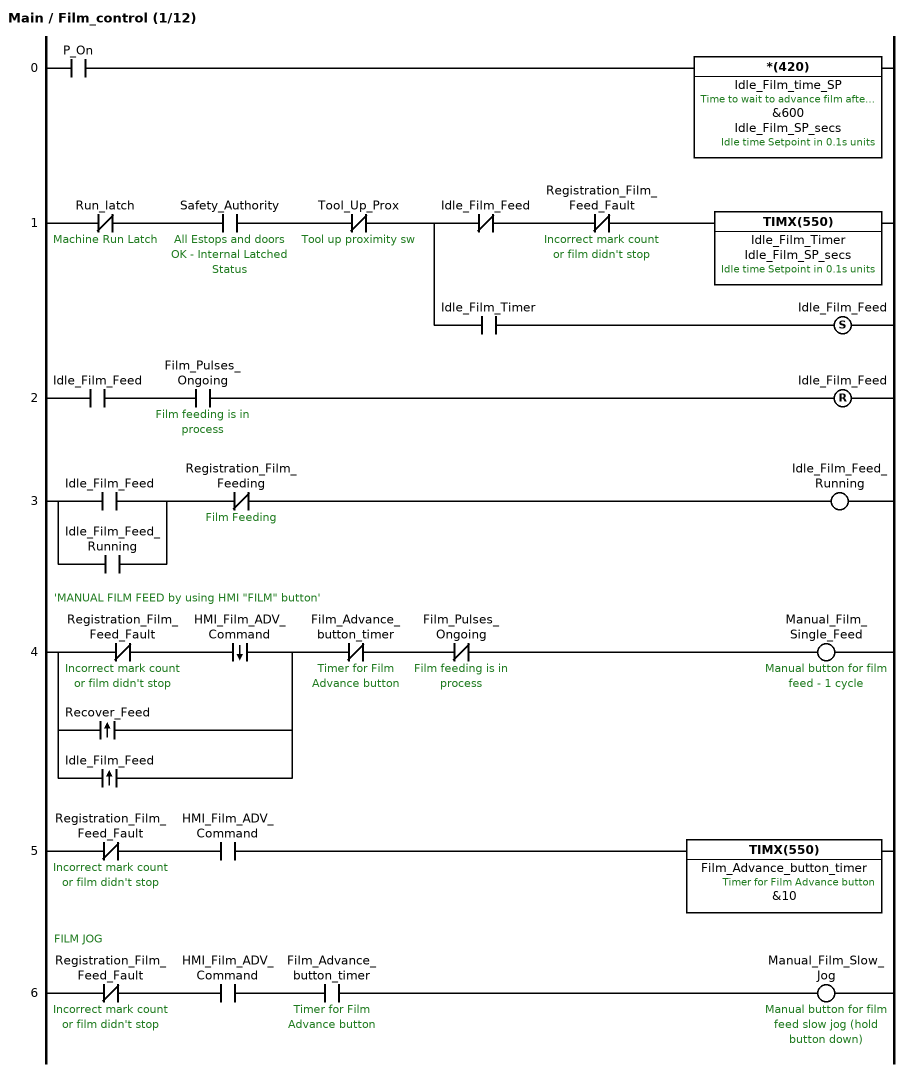
; [picture p72: Main / Film_control, rungs 0-6]
; rung 0
LD P_On
*(420) Idle_Film_time_SP &600 Idle_Film_SP_secs  ; Time to wait to advance film after sitting idle in minutes, Idle time Setpoint in 0.1s units
; rung 1
LDNOT Run_latch  ; Machine Run Latch
AND Safety_Authority  ; All Estops and doors OK - Internal Latched Status
ANDNOT Tool_Up_Prox  ; Tool up proximity sw
OUT TR0
ANDNOT Idle_Film_Feed
ANDNOT Registration_Film_Feed_Fault  ; Incorrect mark count or film didn't stop
TIMX(550) Idle_Film_Timer Idle_Film_SP_secs  ; Idle time Setpoint in 0.1s units
LD TR0
AND Idle_Film_Timer
SET Idle_Film_Feed
; rung 2
LD Idle_Film_Feed
AND Film_Pulses_Ongoing  ; Film feeding is in process
RSET Idle_Film_Feed
; rung 3
LD Idle_Film_Feed
OR Idle_Film_Feed_Running
ANDNOT Registration_Film_Feeding  ; Film Feeding
OUT Idle_Film_Feed_Running
; rung 4: 'MANUAL FILM FEED by using HMI "FILM" button'
LDNOT Registration_Film_Feed_Fault  ; Incorrect mark count or film didn't stop
%AND HMI_Film_ADV_Command
@OR Recover_Feed
@OR Idle_Film_Feed
ANDNOT Film_Advance_button_timer  ; Timer for Film Advance button
ANDNOT Film_Pulses_Ongoing  ; Film feeding is in process
OUT Manual_Film_Single_Feed  ; Manual button for film feed - 1 cycle
; rung 5
LDNOT Registration_Film_Feed_Fault  ; Incorrect mark count or film didn't stop
AND HMI_Film_ADV_Command
TIMX(550) Film_Advance_button_timer &10  ; Timer for Film Advance button
; rung 6: FILM JOG
LDNOT Registration_Film_Feed_Fault  ; Incorrect mark count or film didn't stop
AND HMI_Film_ADV_Command
AND Film_Advance_button_timer  ; Timer for Film Advance button
OUT Manual_Film_Slow_Jog  ; Manual button for film feed slow jog (hold button down)

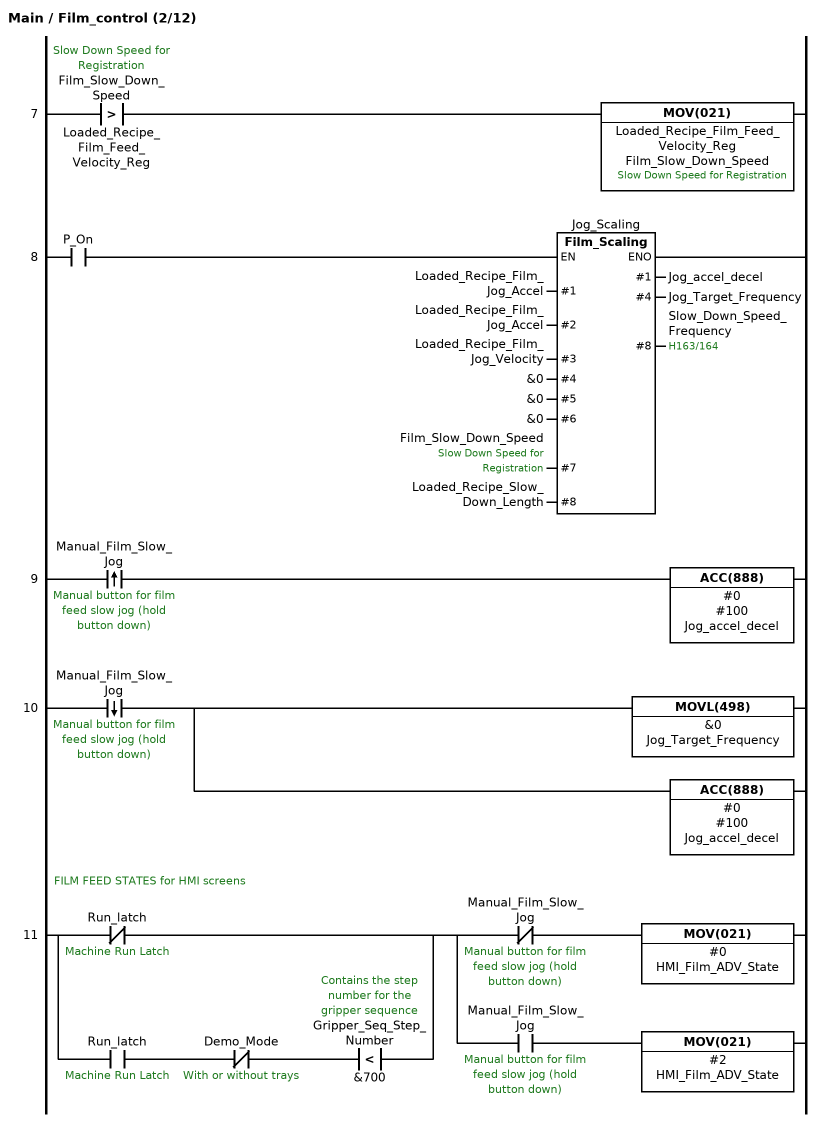
; rung 7
LD>(320) Film_Slow_Down_Speed Loaded_Recipe_Film_Feed_Velocity_Reg  ; Slow Down Speed for Registration
MOV(021) Loaded_Recipe_Film_Feed_Velocity_Reg Film_Slow_Down_Speed  ; Slow Down Speed for Registration
; rung 8
LD P_On
CALL Jog_Scaling : Film_Scaling (#1 := Loaded_Recipe_Film_Jog_Accel, #2 := Loaded_Recipe_Film_Jog_Accel, #3 := Loaded_Recipe_Film_Jog_Velocity, #4 := &0, #5 := &0, #6 := &0, #7 := Film_Slow_Down_Speed, #8 := Loaded_Recipe_Slow_Down_Length)  ; Slow Down Speed for Registration, H163/164
; rung 9
@LD Manual_Film_Slow_Jog  ; Manual button for film feed slow jog (hold button down)
ACC(888) #0 #100 Jog_accel_decel
; rung 10
%LD Manual_Film_Slow_Jog  ; Manual button for film feed slow jog (hold button down)
MOVL(498) &0 Jog_Target_Frequency
ACC(888) #0 #100 Jog_accel_decel
; rung 11: FILM FEED STATES for HMI screens
LDNOT Run_latch  ; Machine Run Latch
LD Run_latch  ; Machine Run Latch
ANDNOT Demo_Mode  ; With or without trays
AND<(310) Gripper_Seq_Step_Number &700  ; Contains the step number for the gripper sequence
ORLD
OUT TR0
ANDNOT Manual_Film_Slow_Jog  ; Manual button for film feed slow jog (hold button down)
MOV(021) #0 HMI_Film_ADV_State
LD TR0
AND Manual_Film_Slow_Jog  ; Manual button for film feed slow jog (hold button down)
MOV(021) #2 HMI_Film_ADV_State

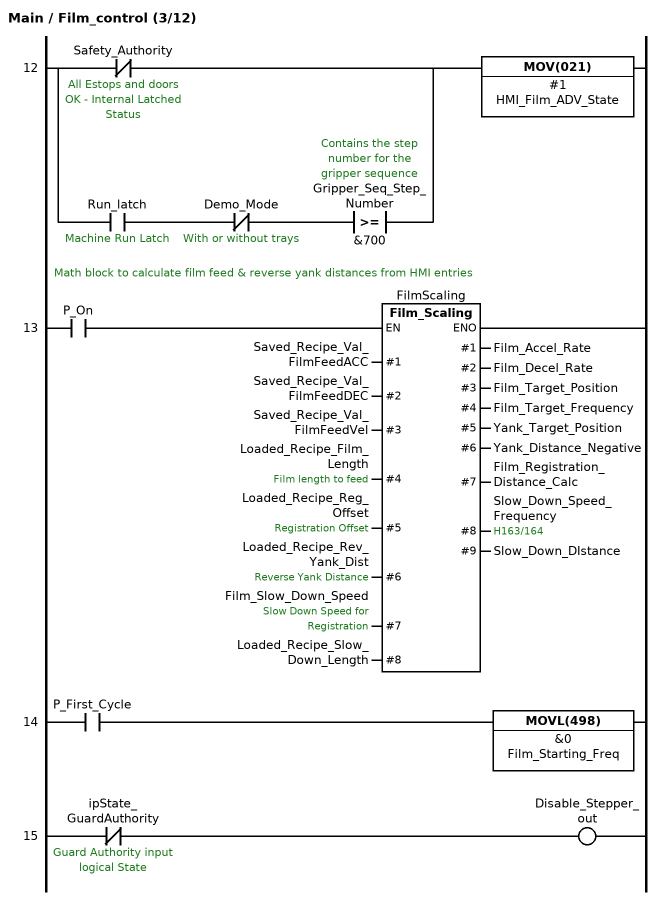
; rung 12
LDNOT Safety_Authority  ; All Estops and doors OK - Internal Latched Status
LD Run_latch  ; Machine Run Latch
ANDNOT Demo_Mode  ; With or without trays
AND>=(325) Gripper_Seq_Step_Number &700  ; Contains the step number for the gripper sequence
ORLD
MOV(021) #1 HMI_Film_ADV_State
; rung 13: Math block to calculate film feed & reverse yank distances from HMI entries
LD P_On
CALL FilmScaling : Film_Scaling (#1 := Saved_Recipe_Val_FilmFeedACC, #2 := Saved_Recipe_Val_FilmFeedDEC, #3 := Saved_Recipe_Val_FilmFeedVel, #4 := Loaded_Recipe_Film_Length, #5 := Loaded_Recipe_Reg_Offset, #6 := Loaded_Recipe_Rev_Yank_Dist, #7 := Film_Slow_Down_Speed, #8 := Loaded_Recipe_Slow_Down_Length, #9 => Slow_Down_DIstance)  ; Film length to feed, Registration Offset, Reverse Yank Distance, Slow Down Speed for Registration, H163/164
; rung 14
LD P_First_Cycle
MOVL(498) &0 Film_Starting_Freq
; rung 15
LDNOT ipState_GuardAuthority  ; Guard Authority input logical State
OUT Disable_Stepper_out

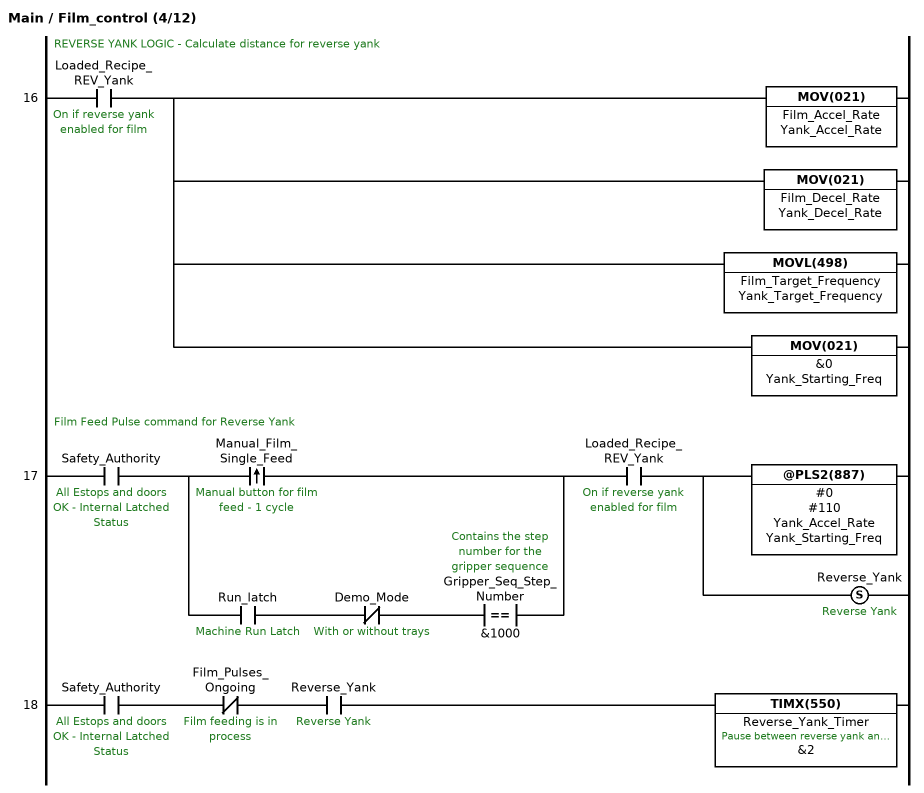
; rung 16: REVERSE YANK LOGIC - Calculate distance for reverse yank
LD Loaded_Recipe_REV_Yank  ; On if reverse yank enabled for film
MOV(021) Film_Accel_Rate Yank_Accel_Rate
MOV(021) Film_Decel_Rate Yank_Decel_Rate
MOVL(498) Film_Target_Frequency Yank_Target_Frequency
MOV(021) &0 Yank_Starting_Freq
; rung 17: Film Feed Pulse command for Reverse Yank
LD Safety_Authority  ; All Estops and doors OK - Internal Latched Status
@LD Manual_Film_Single_Feed  ; Manual button for film feed - 1 cycle
LD Run_latch  ; Machine Run Latch
ANDNOT Demo_Mode  ; With or without trays
AND=(300) Gripper_Seq_Step_Number &1000  ; Contains the step number for the gripper sequence
ORLD
ANDLD
AND Loaded_Recipe_REV_Yank  ; On if reverse yank enabled for film
@PLS2(887) #0 #110 Yank_Accel_Rate Yank_Starting_Freq
SET Reverse_Yank  ; Reverse Yank
; rung 18
LD Safety_Authority  ; All Estops and doors OK - Internal Latched Status
ANDNOT Film_Pulses_Ongoing  ; Film feeding is in process
AND Reverse_Yank  ; Reverse Yank
TIMX(550) Reverse_Yank_Timer &2  ; Pause between reverse yank and moving forward

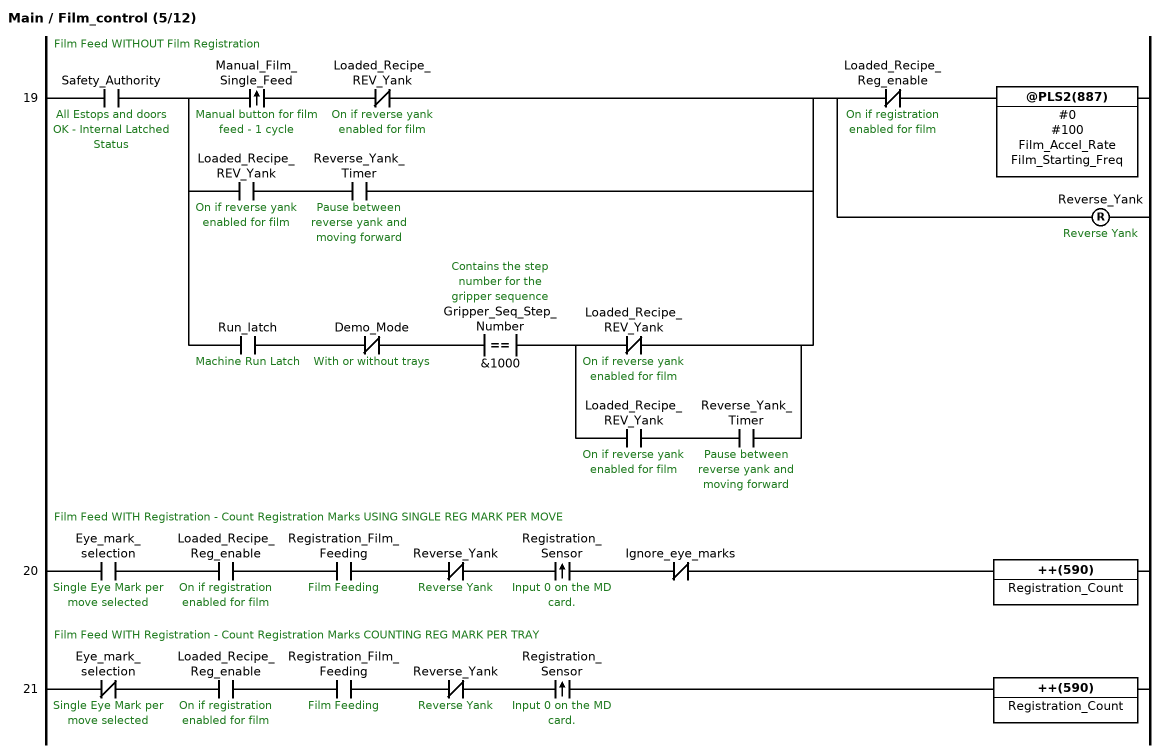
; rung 19: Film Feed WITHOUT Film Registration
LD Safety_Authority  ; All Estops and doors OK - Internal Latched Status
@LD Manual_Film_Single_Feed  ; Manual button for film feed - 1 cycle
ANDNOT Loaded_Recipe_REV_Yank  ; On if reverse yank enabled for film
LD Loaded_Recipe_REV_Yank  ; On if reverse yank enabled for film
AND Reverse_Yank_Timer  ; Pause between reverse yank and moving forward
ORLD
LD Run_latch  ; Machine Run Latch
ANDNOT Demo_Mode  ; With or without trays
AND=(300) Gripper_Seq_Step_Number &1000  ; Contains the step number for the gripper sequence
LDNOT Loaded_Recipe_REV_Yank  ; On if reverse yank enabled for film
LD Loaded_Recipe_REV_Yank  ; On if reverse yank enabled for film
AND Reverse_Yank_Timer  ; Pause between reverse yank and moving forward
ORLD
ANDLD
ORLD
ANDLD
OUT TR0
ANDNOT Loaded_Recipe_Reg_enable  ; On if registration enabled for film
@PLS2(887) #0 #100 Film_Accel_Rate Film_Starting_Freq
LD TR0
RSET Reverse_Yank  ; Reverse Yank
; rung 20: Film Feed WITH Registration - Count Registration Marks USING SINGLE REG MARK PER MOVE
LD Eye_mark_selection  ; Single Eye Mark per move selected
AND Loaded_Recipe_Reg_enable  ; On if registration enabled for film
AND Registration_Film_Feeding  ; Film Feeding
ANDNOT Reverse_Yank  ; Reverse Yank
@AND Registration_Sensor  ; Input 0 on the MD card.
ANDNOT Ignore_eye_marks
++(590) Registration_Count
; rung 21: Film Feed WITH Registration - Count Registration Marks COUNTING REG MARK PER TRAY
LDNOT Eye_mark_selection  ; Single Eye Mark per move selected
AND Loaded_Recipe_Reg_enable  ; On if registration enabled for film
AND Registration_Film_Feeding  ; Film Feeding
ANDNOT Reverse_Yank  ; Reverse Yank
@AND Registration_Sensor  ; Input 0 on the MD card.
++(590) Registration_Count

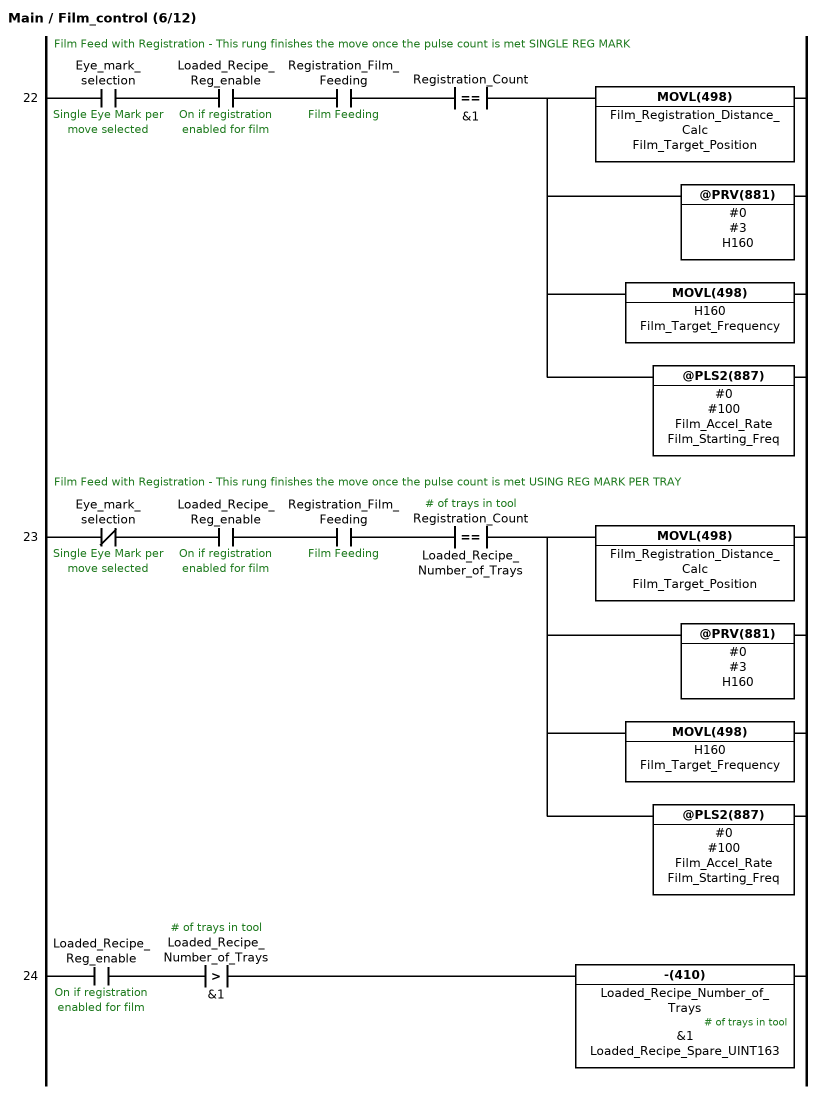
; rung 22: Film Feed with Registration - This rung finishes the move once the pulse count is met SINGLE REG MARK
LD Eye_mark_selection  ; Single Eye Mark per move selected
AND Loaded_Recipe_Reg_enable  ; On if registration enabled for film
AND Registration_Film_Feeding  ; Film Feeding
AND=(300) Registration_Count &1
MOVL(498) Film_Registration_Distance_Calc Film_Target_Position
@PRV(881) #0 #3 H160
MOVL(498) H160 Film_Target_Frequency
@PLS2(887) #0 #100 Film_Accel_Rate Film_Starting_Freq
; rung 23: Film Feed with Registration - This rung finishes the move once the pulse count is met USING REG MARK PER TRAY
LDNOT Eye_mark_selection  ; Single Eye Mark per move selected
AND Loaded_Recipe_Reg_enable  ; On if registration enabled for film
AND Registration_Film_Feeding  ; Film Feeding
AND=(300) Registration_Count Loaded_Recipe_Number_of_Trays  ; # of trays in tool
MOVL(498) Film_Registration_Distance_Calc Film_Target_Position
@PRV(881) #0 #3 H160
MOVL(498) H160 Film_Target_Frequency
@PLS2(887) #0 #100 Film_Accel_Rate Film_Starting_Freq
; rung 24
LD Loaded_Recipe_Reg_enable  ; On if registration enabled for film
AND>(320) Loaded_Recipe_Number_of_Trays &1  ; # of trays in tool
-(410) Loaded_Recipe_Number_of_Trays &1 Loaded_Recipe_Spare_UINT163  ; # of trays in tool

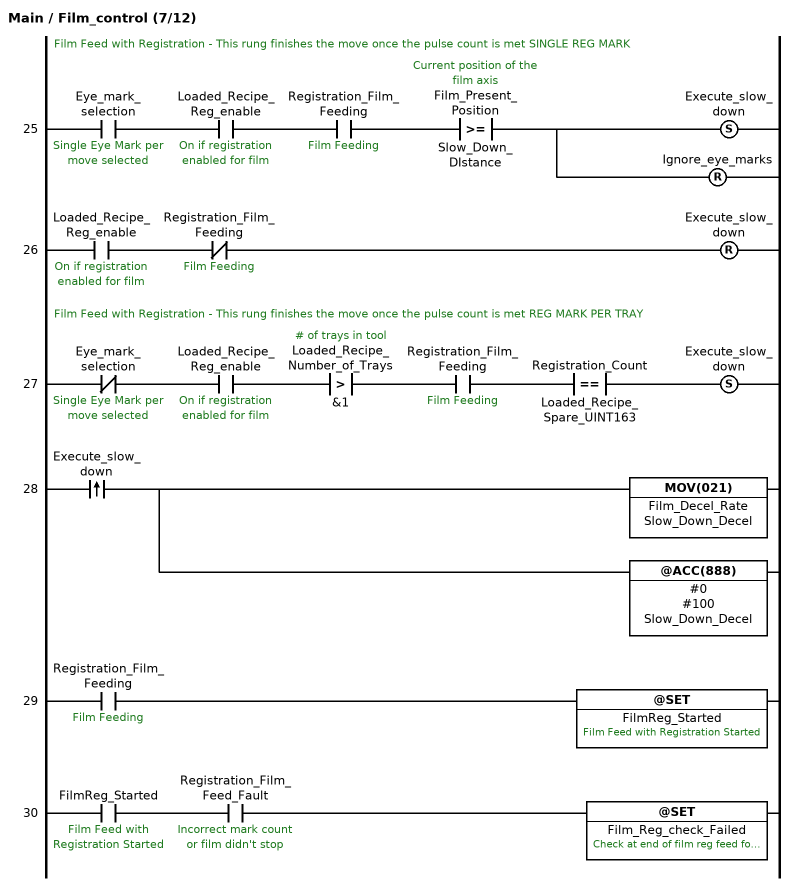
; rung 25: Film Feed with Registration - This rung finishes the move once the pulse count is met SINGLE REG MARK
LD Eye_mark_selection  ; Single Eye Mark per move selected
AND Loaded_Recipe_Reg_enable  ; On if registration enabled for film
AND Registration_Film_Feeding  ; Film Feeding
AND>=(325) Film_Present_Position Slow_Down_DIstance  ; Current position of the film axis
SET Execute_slow_down
RSET Ignore_eye_marks
; rung 26
LD Loaded_Recipe_Reg_enable  ; On if registration enabled for film
ANDNOT Registration_Film_Feeding  ; Film Feeding
RSET Execute_slow_down
; rung 27: Film Feed with Registration - This rung finishes the move once the pulse count is met REG MARK PER TRAY
LDNOT Eye_mark_selection  ; Single Eye Mark per move selected
AND Loaded_Recipe_Reg_enable  ; On if registration enabled for film
AND>(320) Loaded_Recipe_Number_of_Trays &1  ; # of trays in tool
AND Registration_Film_Feeding  ; Film Feeding
AND=(300) Registration_Count Loaded_Recipe_Spare_UINT163
SET Execute_slow_down
; rung 28
@LD Execute_slow_down
MOV(021) Film_Decel_Rate Slow_Down_Decel
@ACC(888) #0 #100 Slow_Down_Decel
; rung 29
LD Registration_Film_Feeding  ; Film Feeding
@SET FilmReg_Started  ; Film Feed with Registration Started
; rung 30
LD FilmReg_Started  ; Film Feed with Registration Started
AND Registration_Film_Feed_Fault  ; Incorrect mark count or film didn't stop
@SET Film_Reg_check_Failed  ; Check at end of film reg feed for problems

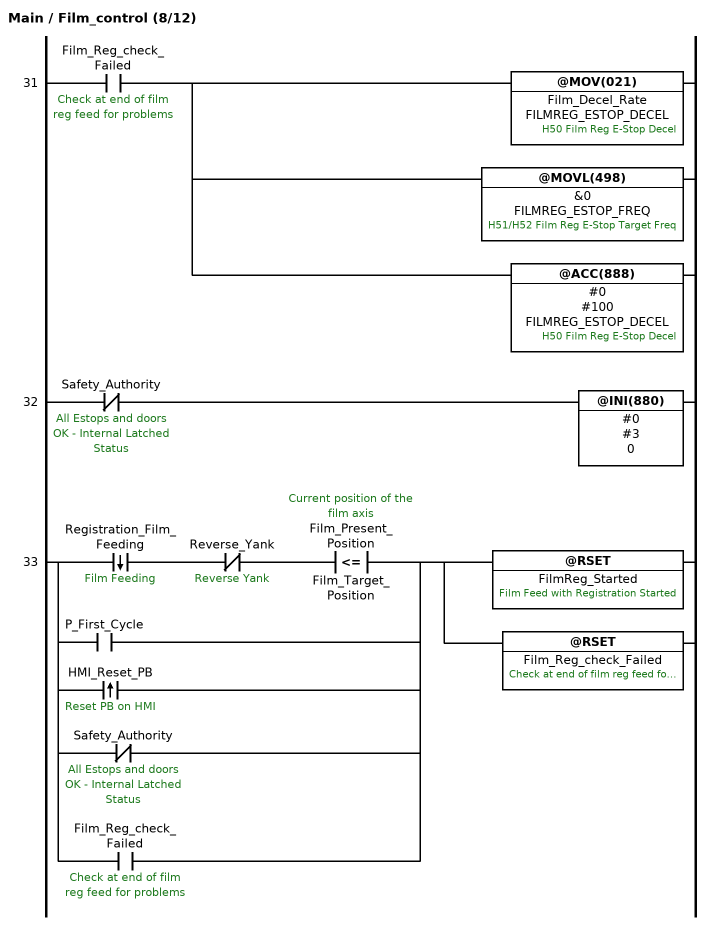
; rung 31
LD Film_Reg_check_Failed  ; Check at end of film reg feed for problems
@MOV(021) Film_Decel_Rate FILMREG_ESTOP_DECEL  ; H50 Film Reg E-Stop Decel
@MOVL(498) &0 FILMREG_ESTOP_FREQ  ; H51/H52 Film Reg E-Stop Target Freq
@ACC(888) #0 #100 FILMREG_ESTOP_DECEL  ; H50 Film Reg E-Stop Decel
; rung 32
LDNOT Safety_Authority  ; All Estops and doors OK - Internal Latched Status
@INI(880) #0 #3 0
; rung 33
%LD Registration_Film_Feeding  ; Film Feeding
ANDNOT Reverse_Yank  ; Reverse Yank
AND<=(315) Film_Present_Position Film_Target_Position  ; Current position of the film axis
OR P_First_Cycle
@OR HMI_Reset_PB  ; Reset PB on HMI
ORNOT Safety_Authority  ; All Estops and doors OK - Internal Latched Status
OR Film_Reg_check_Failed  ; Check at end of film reg feed for problems
@RSET FilmReg_Started  ; Film Feed with Registration Started
@RSET Film_Reg_check_Failed  ; Check at end of film reg feed for problems

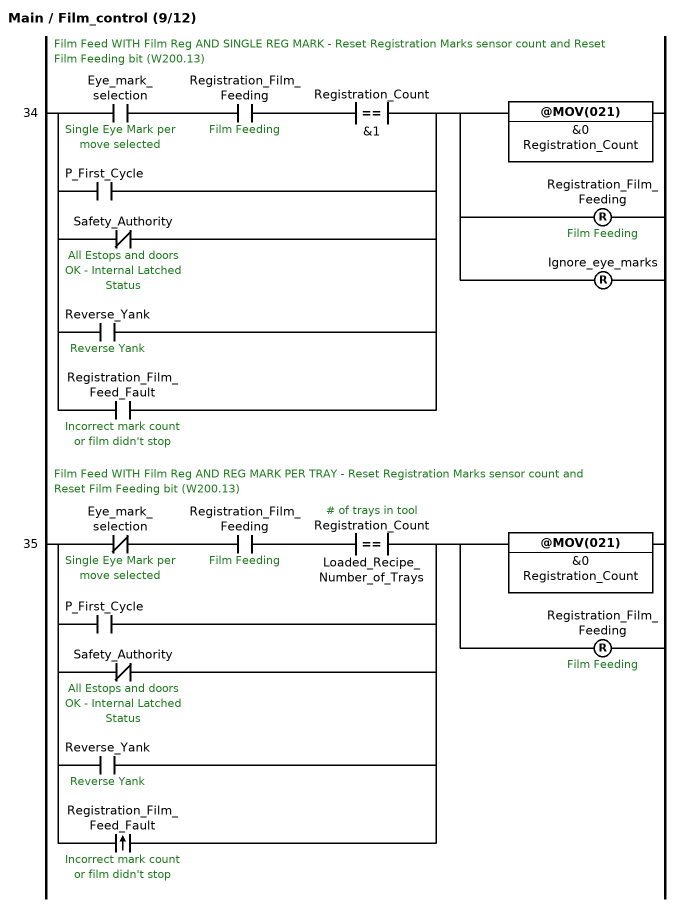
; rung 34: Film Feed WITH Film Reg AND SINGLE REG MARK - Reset Registration Marks sensor count and Reset Film Feeding bit (W200.13)
LD Eye_mark_selection  ; Single Eye Mark per move selected
AND Registration_Film_Feeding  ; Film Feeding
AND=(300) Registration_Count &1
OR P_First_Cycle
ORNOT Safety_Authority  ; All Estops and doors OK - Internal Latched Status
OR Reverse_Yank  ; Reverse Yank
OR Registration_Film_Feed_Fault  ; Incorrect mark count or film didn't stop
@MOV(021) &0 Registration_Count
RSET Registration_Film_Feeding  ; Film Feeding
RSET Ignore_eye_marks
; rung 35: Film Feed WITH Film Reg AND REG MARK PER TRAY - Reset Registration Marks sensor count and Reset Film Feeding bit (W200.13)
LDNOT Eye_mark_selection  ; Single Eye Mark per move selected
AND Registration_Film_Feeding  ; Film Feeding
AND=(300) Registration_Count Loaded_Recipe_Number_of_Trays  ; # of trays in tool
OR P_First_Cycle
ORNOT Safety_Authority  ; All Estops and doors OK - Internal Latched Status
OR Reverse_Yank  ; Reverse Yank
@OR Registration_Film_Feed_Fault  ; Incorrect mark count or film didn't stop
@MOV(021) &0 Registration_Count
RSET Registration_Film_Feeding  ; Film Feeding

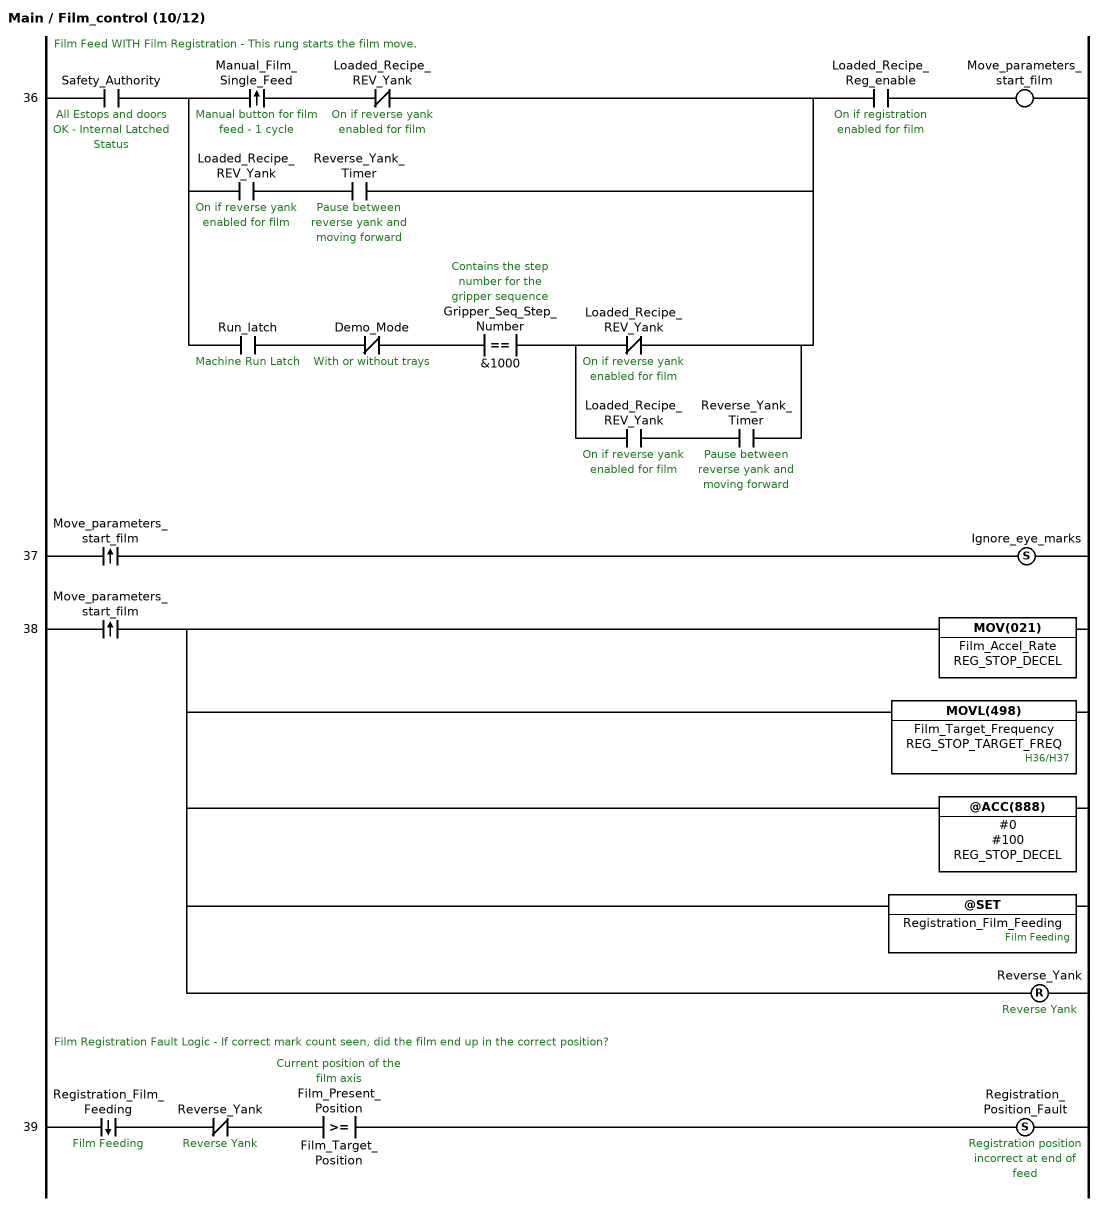
; rung 36: Film Feed WITH Film Registration - This rung starts the film move.
LD Safety_Authority  ; All Estops and doors OK - Internal Latched Status
@LD Manual_Film_Single_Feed  ; Manual button for film feed - 1 cycle
ANDNOT Loaded_Recipe_REV_Yank  ; On if reverse yank enabled for film
LD Loaded_Recipe_REV_Yank  ; On if reverse yank enabled for film
AND Reverse_Yank_Timer  ; Pause between reverse yank and moving forward
ORLD
LD Run_latch  ; Machine Run Latch
ANDNOT Demo_Mode  ; With or without trays
AND=(300) Gripper_Seq_Step_Number &1000  ; Contains the step number for the gripper sequence
LDNOT Loaded_Recipe_REV_Yank  ; On if reverse yank enabled for film
LD Loaded_Recipe_REV_Yank  ; On if reverse yank enabled for film
AND Reverse_Yank_Timer  ; Pause between reverse yank and moving forward
ORLD
ANDLD
ORLD
ANDLD
AND Loaded_Recipe_Reg_enable  ; On if registration enabled for film
OUT Move_parameters_start_film
; rung 37
@LD Move_parameters_start_film
SET Ignore_eye_marks
; rung 38
@LD Move_parameters_start_film
MOV(021) Film_Accel_Rate REG_STOP_DECEL
MOVL(498) Film_Target_Frequency REG_STOP_TARGET_FREQ  ; H36/H37
@ACC(888) #0 #100 REG_STOP_DECEL
@SET Registration_Film_Feeding  ; Film Feeding
RSET Reverse_Yank  ; Reverse Yank
; rung 39: Film Registration Fault Logic - If correct mark count seen, did the film end up in the correct position?
%LD Registration_Film_Feeding  ; Film Feeding
ANDNOT Reverse_Yank  ; Reverse Yank
AND>=(325) Film_Present_Position Film_Target_Position  ; Current position of the film axis
SET Registration_Position_Fault  ; Registration position incorrect at end of feed

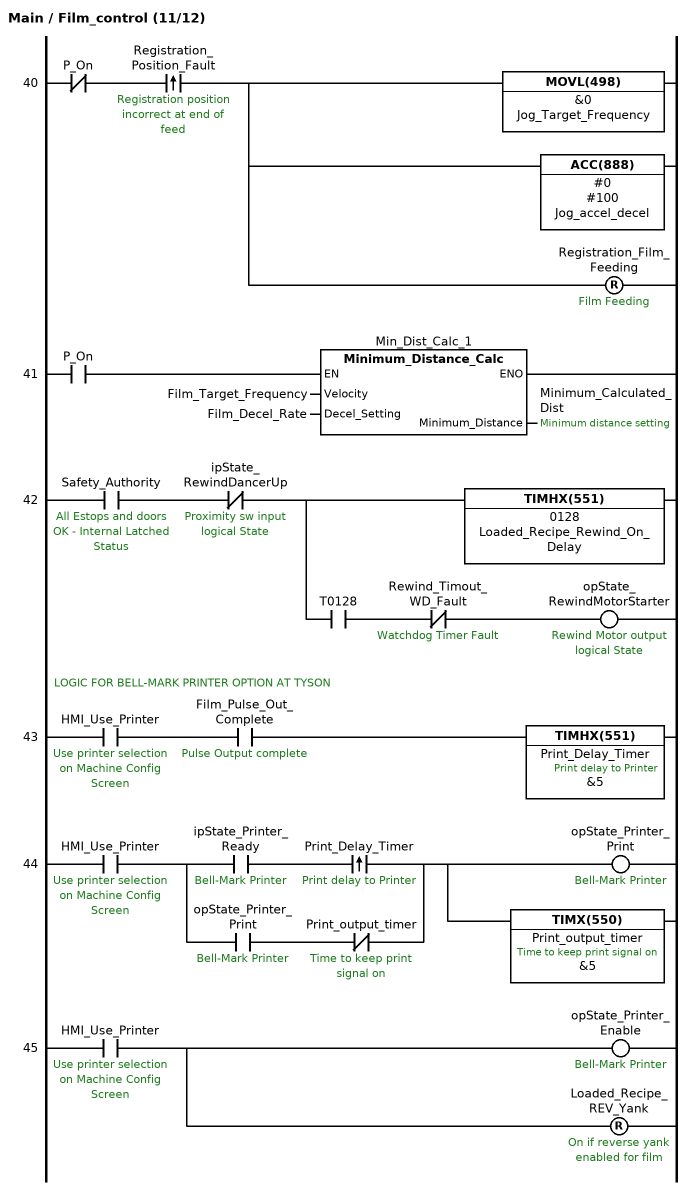
; rung 40
LDNOT P_On
@AND Registration_Position_Fault  ; Registration position incorrect at end of feed
MOVL(498) &0 Jog_Target_Frequency
ACC(888) #0 #100 Jog_accel_decel
RSET Registration_Film_Feeding  ; Film Feeding
; rung 41
LD P_On
CALL Min_Dist_Calc_1 : Minimum_Distance_Calc (Velocity := Film_Target_Frequency, Decel_Setting := Film_Decel_Rate, Minimum_Distance => Minimum_Calculated_Dist)  ; Minimum distance setting
; rung 42
LD Safety_Authority  ; All Estops and doors OK - Internal Latched Status
ANDNOT ipState_RewindDancerUp  ; Proximity sw input logical State
TIMHX(551) 0128 Loaded_Recipe_Rewind_On_Delay
AND T0128
ANDNOT Rewind_Timout_WD_Fault  ; Watchdog Timer Fault
OUT opState_RewindMotorStarter  ; Rewind Motor output logical State
; rung 43: LOGIC FOR BELL-MARK PRINTER OPTION AT TYSON
LD HMI_Use_Printer  ; Use printer selection on Machine Config Screen
AND Film_Pulse_Out_Complete  ; Pulse Output complete
TIMHX(551) Print_Delay_Timer &5  ; Print delay to Printer
; rung 44
LD HMI_Use_Printer  ; Use printer selection on Machine Config Screen
LD ipState_Printer_Ready  ; Bell-Mark Printer
@AND Print_Delay_Timer  ; Print delay to Printer
LD opState_Printer_Print  ; Bell-Mark Printer
ANDNOT Print_output_timer  ; Time to keep print signal on
ORLD
ANDLD
OUT opState_Printer_Print  ; Bell-Mark Printer
TIMX(550) Print_output_timer &5  ; Time to keep print signal on
; rung 45
LD HMI_Use_Printer  ; Use printer selection on Machine Config Screen
OUT opState_Printer_Enable  ; Bell-Mark Printer
RSET Loaded_Recipe_REV_Yank  ; On if reverse yank enabled for film

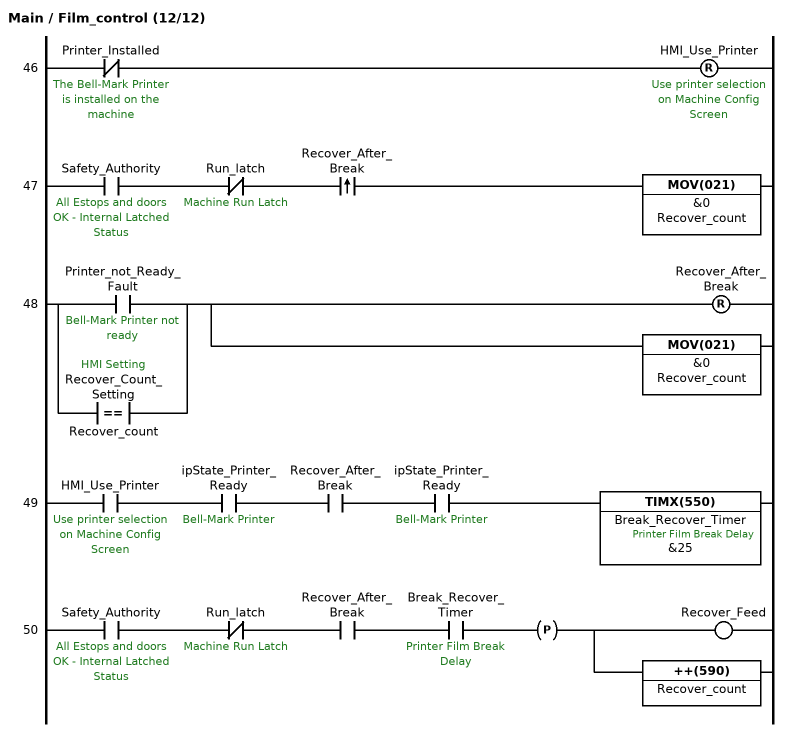
; rung 46
LDNOT Printer_Installed  ; The Bell-Mark Printer is installed on the machine
RSET HMI_Use_Printer  ; Use printer selection on Machine Config Screen
; rung 47
LD Safety_Authority  ; All Estops and doors OK - Internal Latched Status
ANDNOT Run_latch  ; Machine Run Latch
@AND Recover_After_Break
MOV(021) &0 Recover_count
; rung 48
LD Printer_not_Ready_Fault  ; Bell-Mark Printer not ready
OR=(300) Recover_Count_Setting Recover_count  ; HMI Setting
RSET Recover_After_Break
MOV(021) &0 Recover_count
; rung 49
LD HMI_Use_Printer  ; Use printer selection on Machine Config Screen
AND ipState_Printer_Ready  ; Bell-Mark Printer
AND Recover_After_Break
AND ipState_Printer_Ready  ; Bell-Mark Printer
TIMX(550) Break_Recover_Timer &25  ; Printer Film Break Delay
; rung 50
LD Safety_Authority  ; All Estops and doors OK - Internal Latched Status
ANDNOT Run_latch  ; Machine Run Latch
AND Recover_After_Break
AND Break_Recover_Timer  ; Printer Film Break Delay
UP(521)
OUT Recover_Feed
++(590) Recover_count

### Section Watchdog_Timers_and_Faults

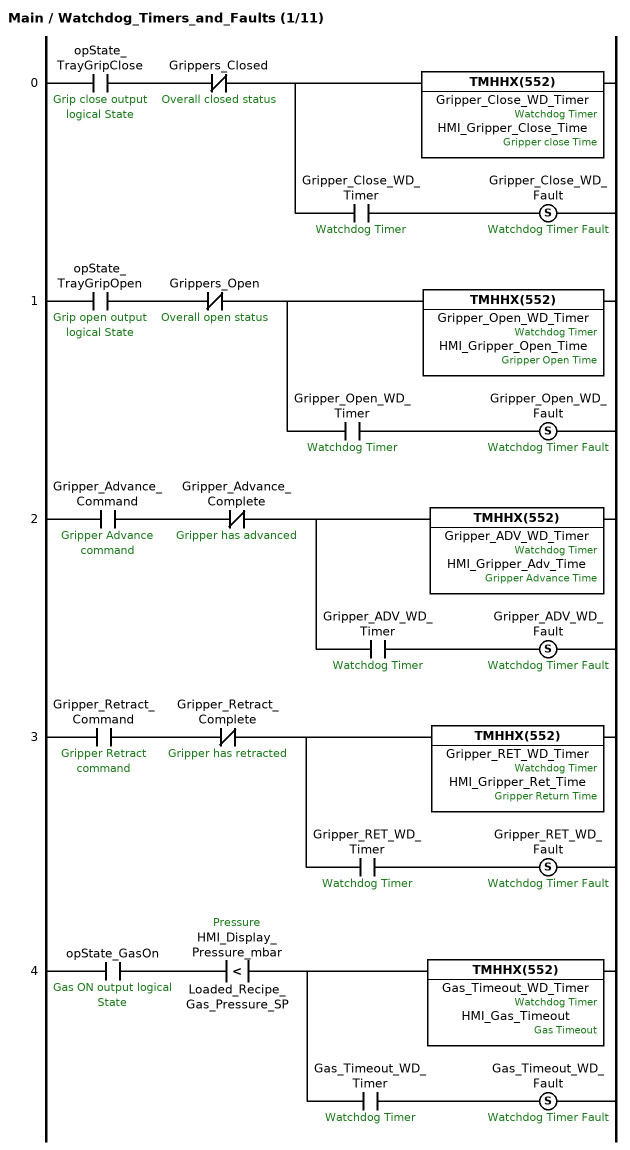
; rung 0
LD opState_TrayGripClose  ; Grip close output logical State
ANDNOT Grippers_Closed  ; Overall closed status
TMHHX(552) Gripper_Close_WD_Timer HMI_Gripper_Close_Time  ; Watchdog Timer, Gripper close Time
AND Gripper_Close_WD_Timer  ; Watchdog Timer
SET Gripper_Close_WD_Fault  ; Watchdog Timer Fault
; rung 1
LD opState_TrayGripOpen  ; Grip open output logical State
ANDNOT Grippers_Open  ; Overall open status
TMHHX(552) Gripper_Open_WD_Timer HMI_Gripper_Open_Time  ; Watchdog Timer, Gripper Open Time
AND Gripper_Open_WD_Timer  ; Watchdog Timer
SET Gripper_Open_WD_Fault  ; Watchdog Timer Fault
; rung 2
LD Gripper_Advance_Command  ; Gripper Advance command
ANDNOT Gripper_Advance_Complete  ; Gripper has advanced
TMHHX(552) Gripper_ADV_WD_Timer HMI_Gripper_Adv_Time  ; Watchdog Timer, Gripper Advance Time
AND Gripper_ADV_WD_Timer  ; Watchdog Timer
SET Gripper_ADV_WD_Fault  ; Watchdog Timer Fault
; rung 3
LD Gripper_Retract_Command  ; Gripper Retract command
ANDNOT Gripper_Retract_Complete  ; Gripper has retracted
TMHHX(552) Gripper_RET_WD_Timer HMI_Gripper_Ret_Time  ; Watchdog Timer, Gripper Return Time
AND Gripper_RET_WD_Timer  ; Watchdog Timer
SET Gripper_RET_WD_Fault  ; Watchdog Timer Fault
; rung 4
LD opState_GasOn  ; Gas ON output logical State
AND<(310) HMI_Display_Pressure_mbar Loaded_Recipe_Gas_Pressure_SP  ; Pressure
TMHHX(552) Gas_Timeout_WD_Timer HMI_Gas_Timeout  ; Watchdog Timer, Gas Timeout
AND Gas_Timeout_WD_Timer  ; Watchdog Timer
SET Gas_Timeout_WD_Fault  ; Watchdog Timer Fault

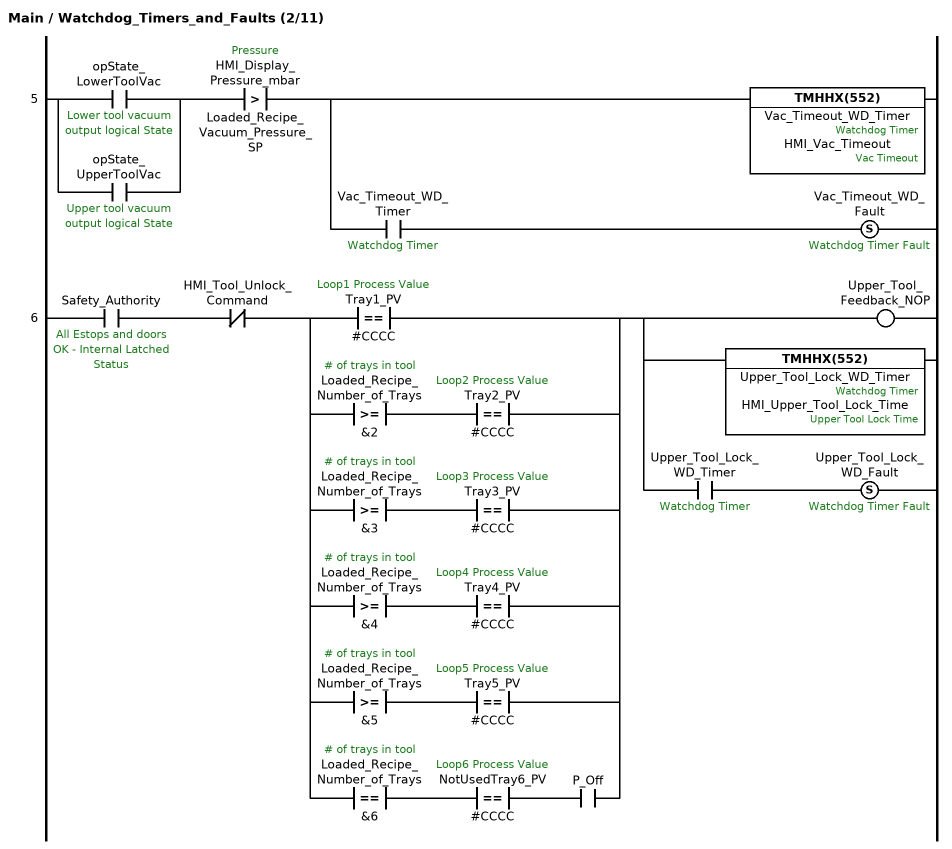
; rung 5
LD opState_LowerToolVac  ; Lower tool vacuum output logical State
OR opState_UpperToolVac  ; Upper tool vacuum output logical State
AND>(320) HMI_Display_Pressure_mbar Loaded_Recipe_Vacuum_Pressure_SP  ; Pressure
TMHHX(552) Vac_Timeout_WD_Timer HMI_Vac_Timeout  ; Watchdog Timer, Vac Timeout
AND Vac_Timeout_WD_Timer  ; Watchdog Timer
SET Vac_Timeout_WD_Fault  ; Watchdog Timer Fault
; rung 6
LD Safety_Authority  ; All Estops and doors OK - Internal Latched Status
ANDNOT HMI_Tool_Unlock_Command
LD=S(302) Tray1_PV #CCCC  ; Loop1 Process Value
LD>=(325) Loaded_Recipe_Number_of_Trays &2  ; # of trays in tool
AND=S(302) Tray2_PV #CCCC  ; Loop2 Process Value
ORLD
LD>=(325) Loaded_Recipe_Number_of_Trays &3  ; # of trays in tool
AND=S(302) Tray3_PV #CCCC  ; Loop3 Process Value
ORLD
LD>=(325) Loaded_Recipe_Number_of_Trays &4  ; # of trays in tool
AND=S(302) Tray4_PV #CCCC  ; Loop4 Process Value
ORLD
LD>=(325) Loaded_Recipe_Number_of_Trays &5  ; # of trays in tool
AND=S(302) Tray5_PV #CCCC  ; Loop5 Process Value
ORLD
LD=(300) Loaded_Recipe_Number_of_Trays &6  ; # of trays in tool
AND=S(302) NotUsedTray6_PV #CCCC  ; Loop6 Process Value
AND P_Off
ORLD
ANDLD
OUT Upper_Tool_Feedback_NOP
TMHHX(552) Upper_Tool_Lock_WD_Timer HMI_Upper_Tool_Lock_Time  ; Watchdog Timer, Upper Tool Lock Time
AND Upper_Tool_Lock_WD_Timer  ; Watchdog Timer
SET Upper_Tool_Lock_WD_Fault  ; Watchdog Timer Fault

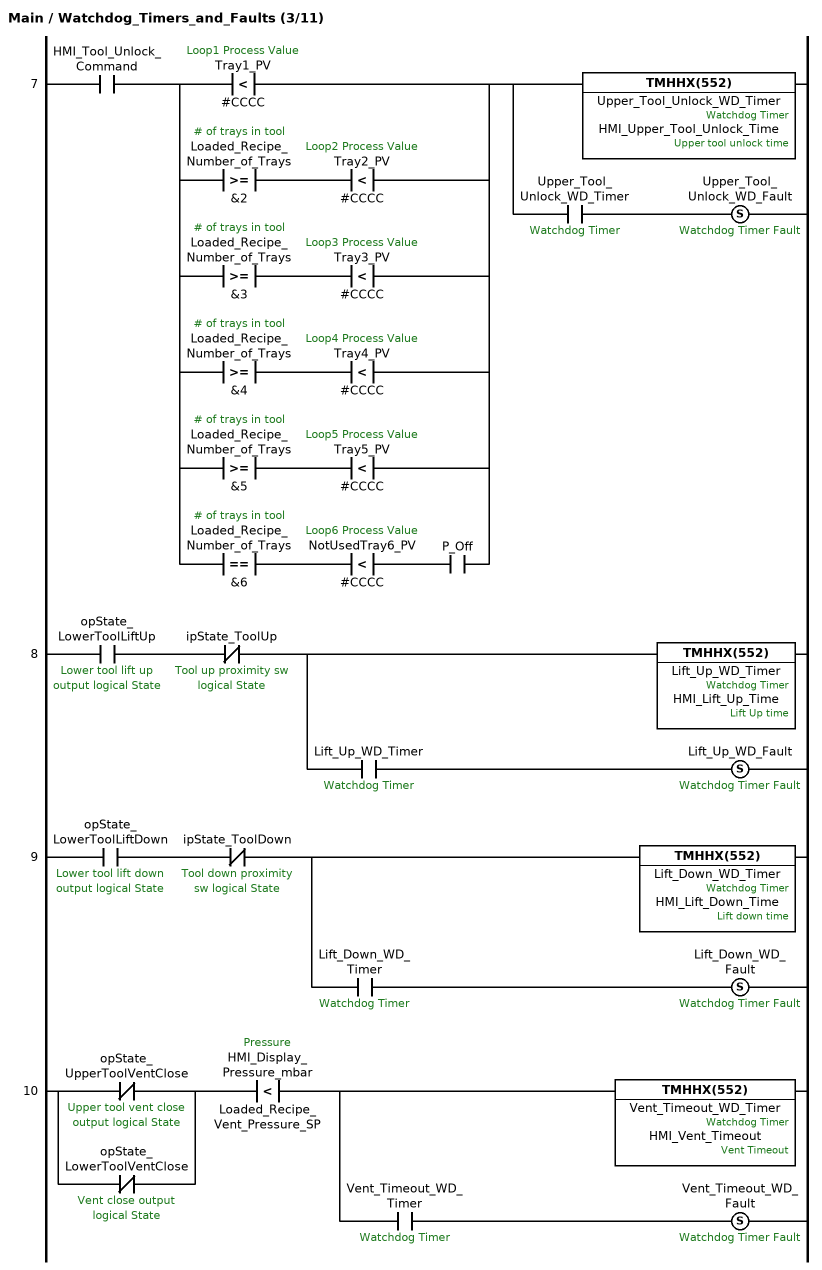
; rung 7
LD HMI_Tool_Unlock_Command
LD<S(312) Tray1_PV #CCCC  ; Loop1 Process Value
LD>=(325) Loaded_Recipe_Number_of_Trays &2  ; # of trays in tool
AND<S(312) Tray2_PV #CCCC  ; Loop2 Process Value
ORLD
LD>=(325) Loaded_Recipe_Number_of_Trays &3  ; # of trays in tool
AND<S(312) Tray3_PV #CCCC  ; Loop3 Process Value
ORLD
LD>=(325) Loaded_Recipe_Number_of_Trays &4  ; # of trays in tool
AND<S(312) Tray4_PV #CCCC  ; Loop4 Process Value
ORLD
LD>=(325) Loaded_Recipe_Number_of_Trays &5  ; # of trays in tool
AND<S(312) Tray5_PV #CCCC  ; Loop5 Process Value
ORLD
LD=(300) Loaded_Recipe_Number_of_Trays &6  ; # of trays in tool
AND<S(312) NotUsedTray6_PV #CCCC  ; Loop6 Process Value
AND P_Off
ORLD
ANDLD
TMHHX(552) Upper_Tool_Unlock_WD_Timer HMI_Upper_Tool_Unlock_Time  ; Watchdog Timer, Upper tool unlock time
AND Upper_Tool_Unlock_WD_Timer  ; Watchdog Timer
SET Upper_Tool_Unlock_WD_Fault  ; Watchdog Timer Fault
; rung 8
LD opState_LowerToolLiftUp  ; Lower tool lift up output logical State
ANDNOT ipState_ToolUp  ; Tool up proximity sw logical State
TMHHX(552) Lift_Up_WD_Timer HMI_Lift_Up_Time  ; Watchdog Timer, Lift Up time
AND Lift_Up_WD_Timer  ; Watchdog Timer
SET Lift_Up_WD_Fault  ; Watchdog Timer Fault
; rung 9
LD opState_LowerToolLiftDown  ; Lower tool lift down output logical State
ANDNOT ipState_ToolDown  ; Tool down proximity sw logical State
TMHHX(552) Lift_Down_WD_Timer HMI_Lift_Down_Time  ; Watchdog Timer, Lift down time
AND Lift_Down_WD_Timer  ; Watchdog Timer
SET Lift_Down_WD_Fault  ; Watchdog Timer Fault
; rung 10
LDNOT opState_UpperToolVentClose  ; Upper tool vent close output logical State
ORNOT opState_LowerToolVentClose  ; Vent close output logical State
AND<(310) HMI_Display_Pressure_mbar Loaded_Recipe_Vent_Pressure_SP  ; Pressure
TMHHX(552) Vent_Timeout_WD_Timer HMI_Vent_Timeout  ; Watchdog Timer, Vent Timeout
AND Vent_Timeout_WD_Timer  ; Watchdog Timer
SET Vent_Timeout_WD_Fault  ; Watchdog Timer Fault

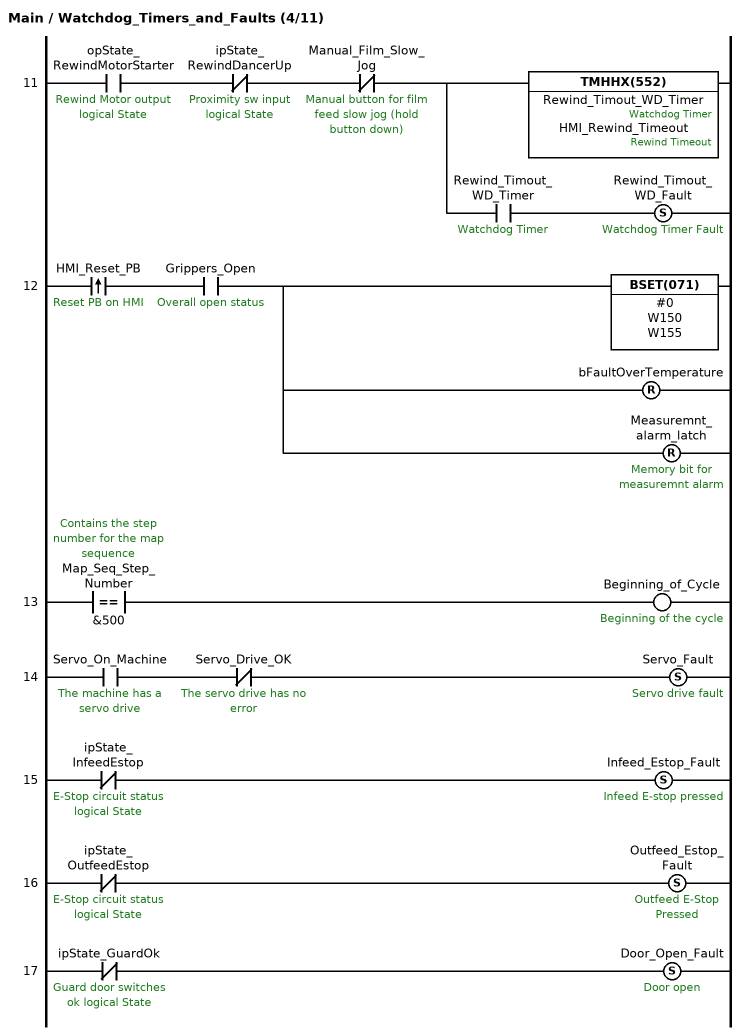
; rung 11
LD opState_RewindMotorStarter  ; Rewind Motor output logical State
ANDNOT ipState_RewindDancerUp  ; Proximity sw input logical State
ANDNOT Manual_Film_Slow_Jog  ; Manual button for film feed slow jog (hold button down)
TMHHX(552) Rewind_Timout_WD_Timer HMI_Rewind_Timeout  ; Watchdog Timer, Rewind Timeout
AND Rewind_Timout_WD_Timer  ; Watchdog Timer
SET Rewind_Timout_WD_Fault  ; Watchdog Timer Fault
; rung 12
@LD HMI_Reset_PB  ; Reset PB on HMI
AND Grippers_Open  ; Overall open status
BSET(071) #0 W150 W155
RSET bFaultOverTemperature
RSET Measuremnt_alarm_latch  ; Memory bit for measuremnt alarm
; rung 13
LD=(300) Map_Seq_Step_Number &500  ; Contains the step number for the map sequence
OUT Beginning_of_Cycle  ; Beginning of the cycle
; rung 14
LD Servo_On_Machine  ; The machine has a servo drive
ANDNOT Servo_Drive_OK  ; The servo drive has no error
SET Servo_Fault  ; Servo drive fault
; rung 15
LDNOT ipState_InfeedEstop  ; E-Stop circuit status logical State
SET Infeed_Estop_Fault  ; Infeed E-stop pressed
; rung 16
LDNOT ipState_OutfeedEstop  ; E-Stop circuit status logical State
SET Outfeed_Estop_Fault  ; Outfeed E-Stop Pressed
; rung 17
LDNOT ipState_GuardOk  ; Guard door switches ok logical State
SET Door_Open_Fault  ; Door open

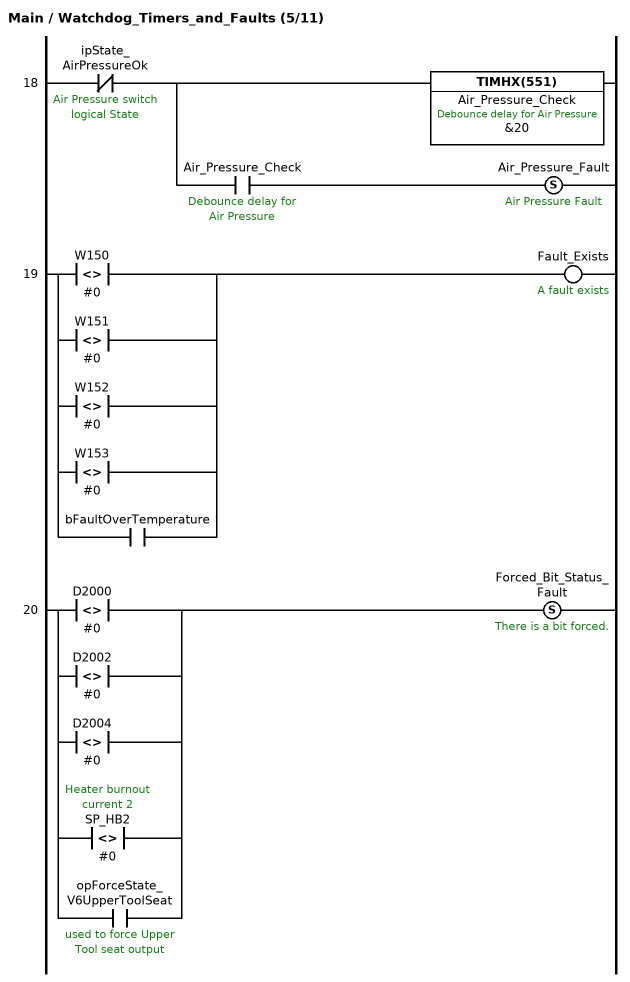
; rung 18
LDNOT ipState_AirPressureOk  ; Air Pressure switch logical State
TIMHX(551) Air_Pressure_Check &20  ; Debounce delay for Air Pressure
AND Air_Pressure_Check  ; Debounce delay for Air Pressure
SET Air_Pressure_Fault  ; Air Pressure Fault
; rung 19
LD<>(305) W150 #0
OR<>(305) W151 #0
OR<>(305) W152 #0
OR<>(305) W153 #0
OR bFaultOverTemperature
OUT Fault_Exists  ; A fault exists
; rung 20
LD<>(305) D2000 #0
OR<>(305) D2002 #0
OR<>(305) D2004 #0
OR<>(305) SP_HB2 #0  ; Heater burnout current 2
OR opForceState_V6UpperToolSeat  ; used to force Upper Tool seat output
SET Forced_Bit_Status_Fault  ; There is a bit forced.

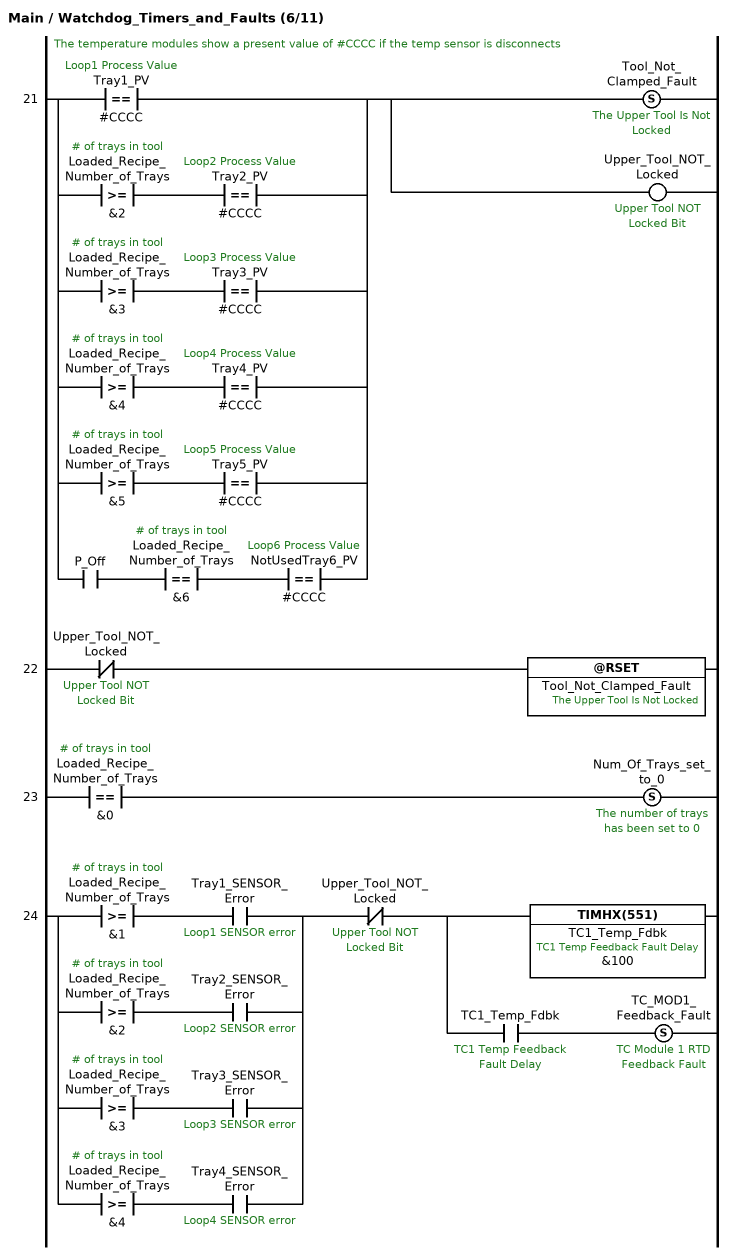
; rung 21: The temperature modules show a present value of #CCCC if the temp sensor is disconnects
LD=S(302) Tray1_PV #CCCC  ; Loop1 Process Value
LD>=(325) Loaded_Recipe_Number_of_Trays &2  ; # of trays in tool
AND=S(302) Tray2_PV #CCCC  ; Loop2 Process Value
ORLD
LD>=(325) Loaded_Recipe_Number_of_Trays &3  ; # of trays in tool
AND=S(302) Tray3_PV #CCCC  ; Loop3 Process Value
ORLD
LD>=(325) Loaded_Recipe_Number_of_Trays &4  ; # of trays in tool
AND=S(302) Tray4_PV #CCCC  ; Loop4 Process Value
ORLD
LD>=(325) Loaded_Recipe_Number_of_Trays &5  ; # of trays in tool
AND=S(302) Tray5_PV #CCCC  ; Loop5 Process Value
ORLD
LD P_Off
AND=(300) Loaded_Recipe_Number_of_Trays &6  ; # of trays in tool
AND=S(302) NotUsedTray6_PV #CCCC  ; Loop6 Process Value
ORLD
SET Tool_Not_Clamped_Fault  ; The Upper Tool Is Not Locked
OUT Upper_Tool_NOT_Locked  ; Upper Tool NOT Locked Bit
; rung 22
LDNOT Upper_Tool_NOT_Locked  ; Upper Tool NOT Locked Bit
@RSET Tool_Not_Clamped_Fault  ; The Upper Tool Is Not Locked
; rung 23
LD=(300) Loaded_Recipe_Number_of_Trays &0  ; # of trays in tool
SET Num_Of_Trays_set_to_0  ; The number of trays has been set to 0
; rung 24
LD>=(325) Loaded_Recipe_Number_of_Trays &1  ; # of trays in tool
AND Tray1_SENSOR_Error  ; Loop1 SENSOR error
LD>=(325) Loaded_Recipe_Number_of_Trays &2  ; # of trays in tool
AND Tray2_SENSOR_Error  ; Loop2 SENSOR error
ORLD
LD>=(325) Loaded_Recipe_Number_of_Trays &3  ; # of trays in tool
AND Tray3_SENSOR_Error  ; Loop3 SENSOR error
ORLD
LD>=(325) Loaded_Recipe_Number_of_Trays &4  ; # of trays in tool
AND Tray4_SENSOR_Error  ; Loop4 SENSOR error
ORLD
ANDNOT Upper_Tool_NOT_Locked  ; Upper Tool NOT Locked Bit
TIMHX(551) TC1_Temp_Fdbk &100  ; TC1 Temp Feedback Fault Delay
AND TC1_Temp_Fdbk  ; TC1 Temp Feedback Fault Delay
SET TC_MOD1_Feedback_Fault  ; TC Module 1 RTD Feedback Fault

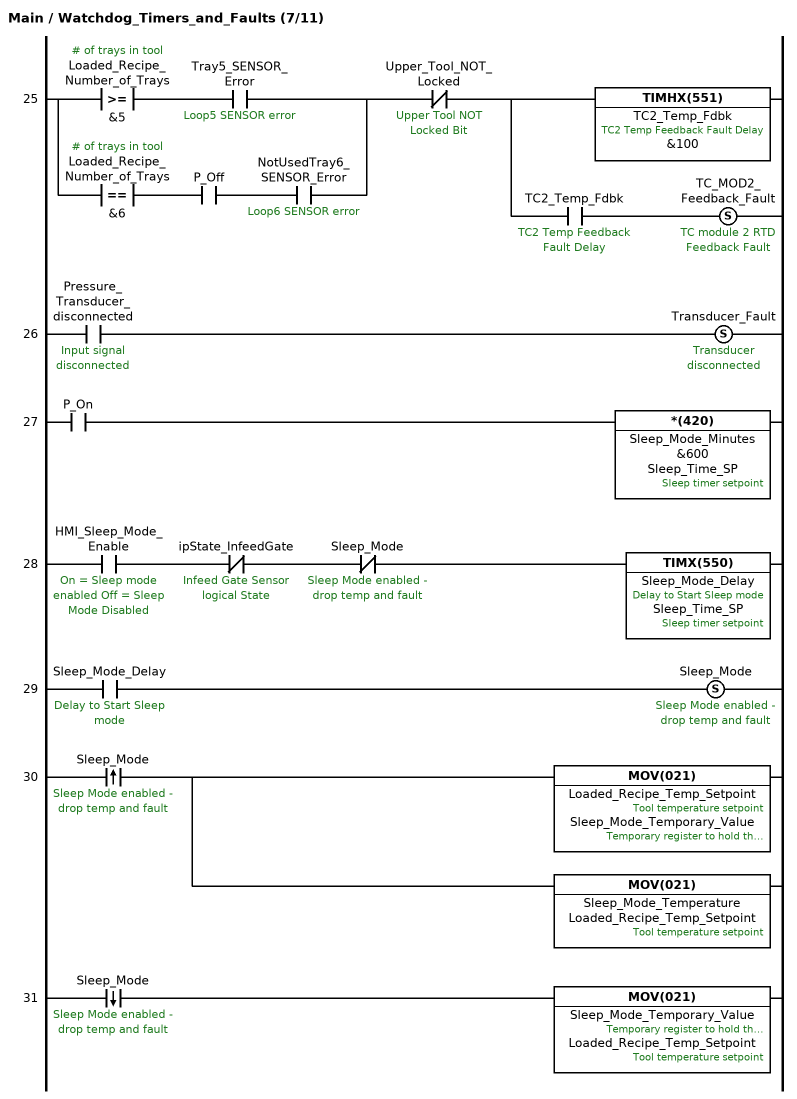
; rung 25
LD>=(325) Loaded_Recipe_Number_of_Trays &5  ; # of trays in tool
AND Tray5_SENSOR_Error  ; Loop5 SENSOR error
LD=(300) Loaded_Recipe_Number_of_Trays &6  ; # of trays in tool
AND P_Off
AND NotUsedTray6_SENSOR_Error  ; Loop6 SENSOR error
ORLD
ANDNOT Upper_Tool_NOT_Locked  ; Upper Tool NOT Locked Bit
TIMHX(551) TC2_Temp_Fdbk &100  ; TC2 Temp Feedback Fault Delay
AND TC2_Temp_Fdbk  ; TC2 Temp Feedback Fault Delay
SET TC_MOD2_Feedback_Fault  ; TC module 2 RTD Feedback Fault
; rung 26
LD Pressure_Transducer_disconnected  ; Input signal disconnected
SET Transducer_Fault  ; Transducer disconnected
; rung 27
LD P_On
*(420) Sleep_Mode_Minutes &600 Sleep_Time_SP  ; Sleep timer setpoint
; rung 28
LD HMI_Sleep_Mode_Enable  ; On = Sleep mode enabled Off = Sleep Mode Disabled
ANDNOT ipState_InfeedGate  ; Infeed Gate Sensor logical State
ANDNOT Sleep_Mode  ; Sleep Mode enabled - drop temp and fault
TIMX(550) Sleep_Mode_Delay Sleep_Time_SP  ; Delay to Start Sleep mode, Sleep timer setpoint
; rung 29
LD Sleep_Mode_Delay  ; Delay to Start Sleep mode
SET Sleep_Mode  ; Sleep Mode enabled - drop temp and fault
; rung 30
@LD Sleep_Mode  ; Sleep Mode enabled - drop temp and fault
MOV(021) Loaded_Recipe_Temp_Setpoint Sleep_Mode_Temporary_Value  ; Tool temperature setpoint, Temporary register to hold the temperature setpoint while in sleep mode
MOV(021) Sleep_Mode_Temperature Loaded_Recipe_Temp_Setpoint  ; Tool temperature setpoint
; rung 31
%LD Sleep_Mode  ; Sleep Mode enabled - drop temp and fault
MOV(021) Sleep_Mode_Temporary_Value Loaded_Recipe_Temp_Setpoint  ; Temporary register to hold the temperature setpoint while in sleep mode, Tool temperature setpoint

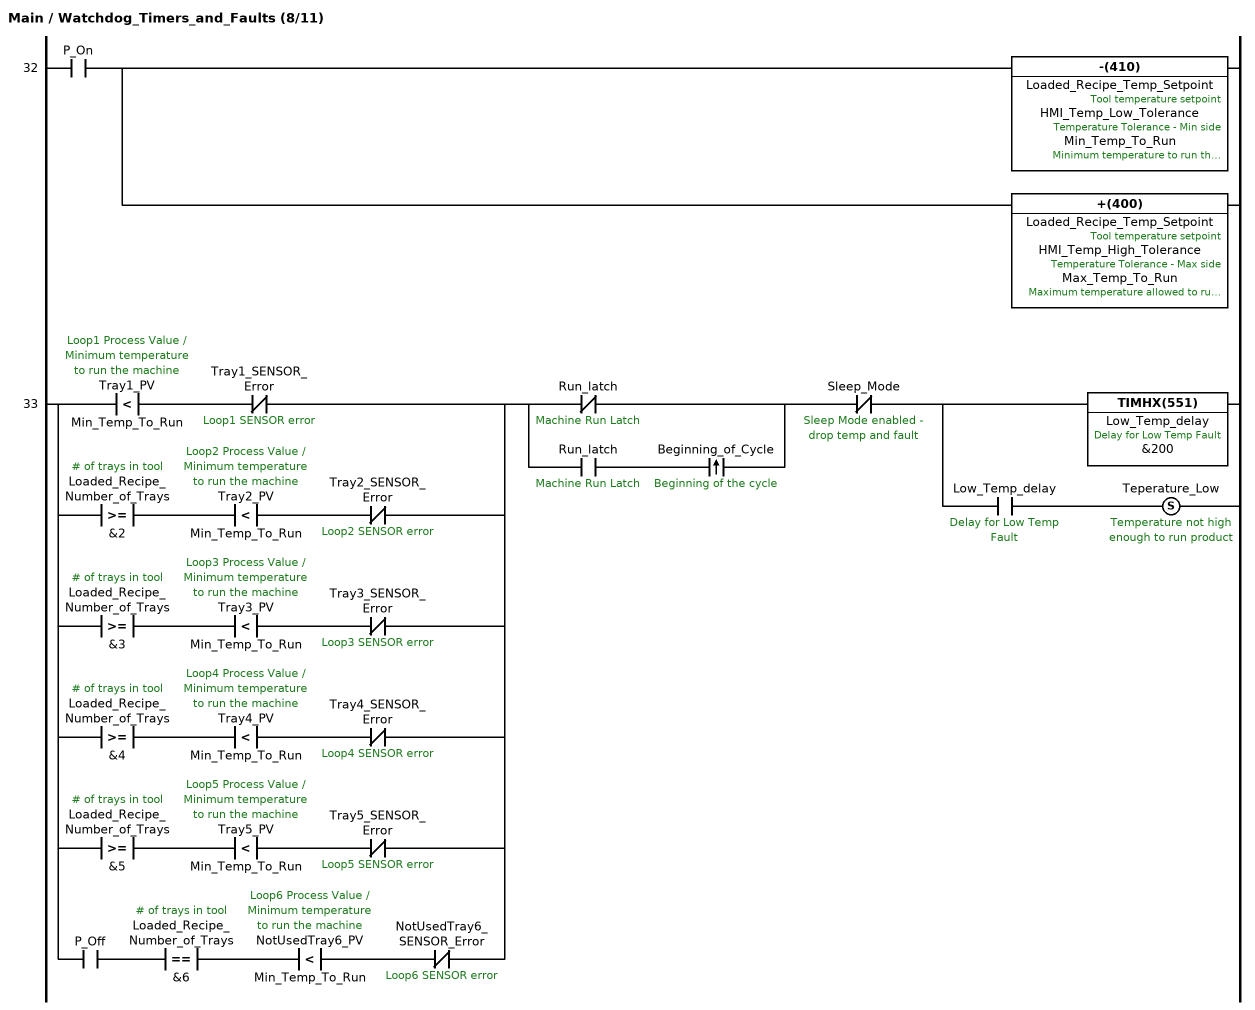
; rung 32
LD P_On
-(410) Loaded_Recipe_Temp_Setpoint HMI_Temp_Low_Tolerance Min_Temp_To_Run  ; Tool temperature setpoint, Temperature Tolerance - Min side, Minimum temperature to run the machine
+(400) Loaded_Recipe_Temp_Setpoint HMI_Temp_High_Tolerance Max_Temp_To_Run  ; Tool temperature setpoint, Temperature Tolerance - Max side, Maximum temperature allowed to run the machine
; rung 33
LD<S(312) Tray1_PV Min_Temp_To_Run  ; Loop1 Process Value, Minimum temperature to run the machine
ANDNOT Tray1_SENSOR_Error  ; Loop1 SENSOR error
LD>=(325) Loaded_Recipe_Number_of_Trays &2  ; # of trays in tool
AND<S(312) Tray2_PV Min_Temp_To_Run  ; Loop2 Process Value, Minimum temperature to run the machine
ANDNOT Tray2_SENSOR_Error  ; Loop2 SENSOR error
ORLD
LD>=(325) Loaded_Recipe_Number_of_Trays &3  ; # of trays in tool
AND<S(312) Tray3_PV Min_Temp_To_Run  ; Loop3 Process Value, Minimum temperature to run the machine
ANDNOT Tray3_SENSOR_Error  ; Loop3 SENSOR error
ORLD
LD>=(325) Loaded_Recipe_Number_of_Trays &4  ; # of trays in tool
AND<S(312) Tray4_PV Min_Temp_To_Run  ; Loop4 Process Value, Minimum temperature to run the machine
ANDNOT Tray4_SENSOR_Error  ; Loop4 SENSOR error
ORLD
LD>=(325) Loaded_Recipe_Number_of_Trays &5  ; # of trays in tool
AND<S(312) Tray5_PV Min_Temp_To_Run  ; Loop5 Process Value, Minimum temperature to run the machine
ANDNOT Tray5_SENSOR_Error  ; Loop5 SENSOR error
ORLD
LD P_Off
AND=(300) Loaded_Recipe_Number_of_Trays &6  ; # of trays in tool
AND<S(312) NotUsedTray6_PV Min_Temp_To_Run  ; Loop6 Process Value, Minimum temperature to run the machine
ANDNOT NotUsedTray6_SENSOR_Error  ; Loop6 SENSOR error
ORLD
LDNOT Run_latch  ; Machine Run Latch
LD Run_latch  ; Machine Run Latch
@AND Beginning_of_Cycle  ; Beginning of the cycle
ORLD
ANDLD
ANDNOT Sleep_Mode  ; Sleep Mode enabled - drop temp and fault
TIMHX(551) Low_Temp_delay &200  ; Delay for Low Temp Fault
AND Low_Temp_delay  ; Delay for Low Temp Fault
SET Teperature_Low  ; Temperature not high enough to run product

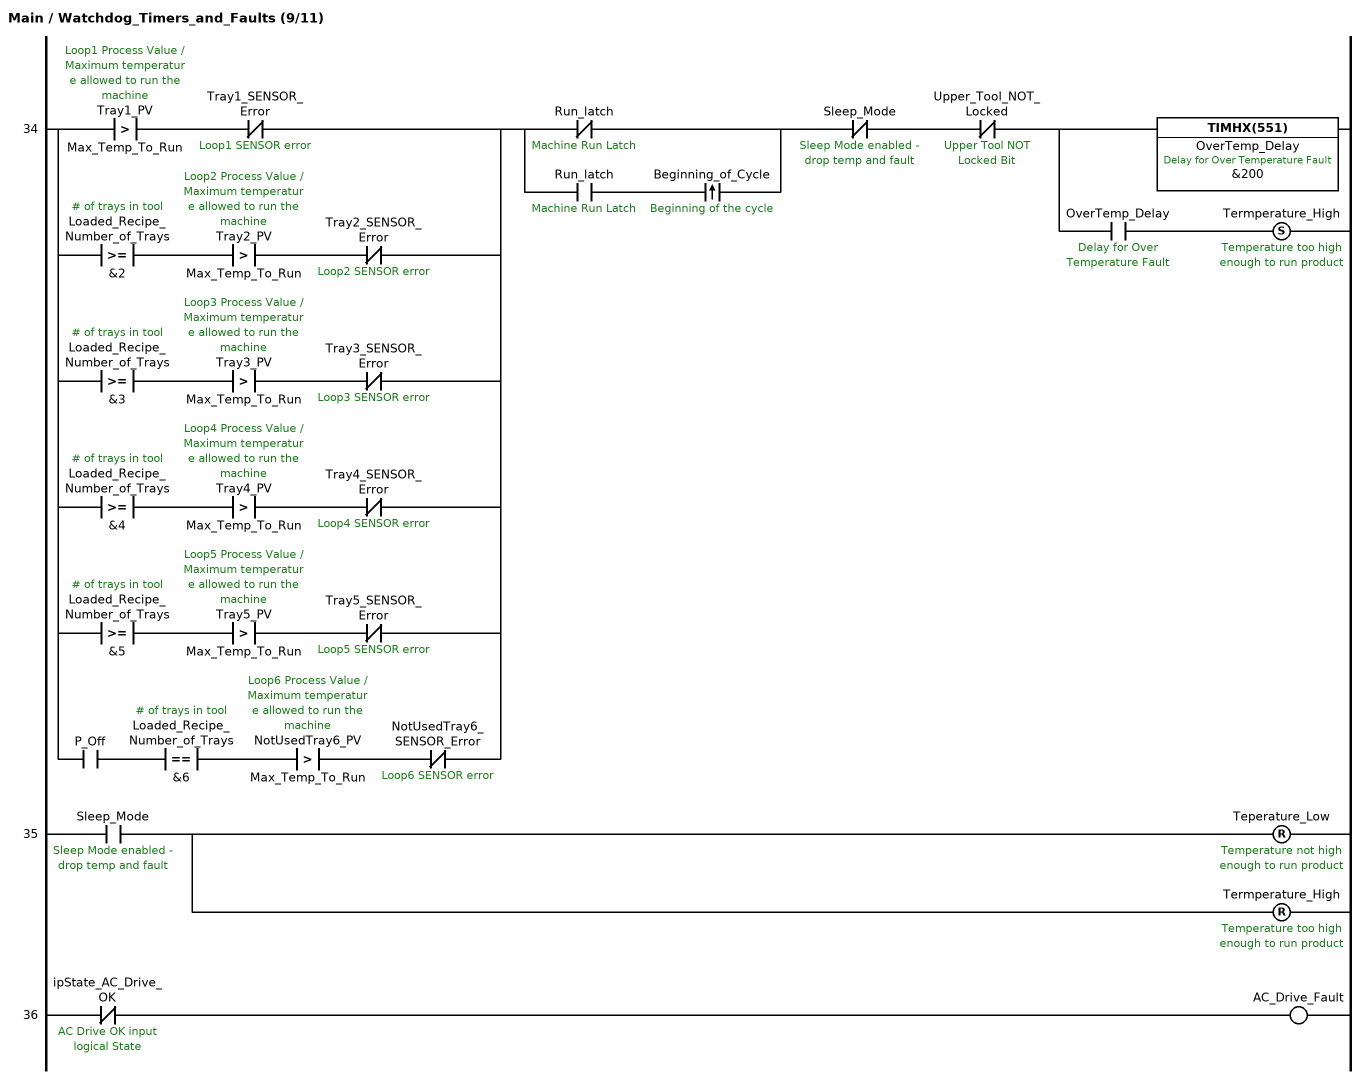
; rung 34
LD>S(322) Tray1_PV Max_Temp_To_Run  ; Loop1 Process Value, Maximum temperature allowed to run the machine
ANDNOT Tray1_SENSOR_Error  ; Loop1 SENSOR error
LD>=(325) Loaded_Recipe_Number_of_Trays &2  ; # of trays in tool
AND>S(322) Tray2_PV Max_Temp_To_Run  ; Loop2 Process Value, Maximum temperature allowed to run the machine
ANDNOT Tray2_SENSOR_Error  ; Loop2 SENSOR error
ORLD
LD>=(325) Loaded_Recipe_Number_of_Trays &3  ; # of trays in tool
AND>S(322) Tray3_PV Max_Temp_To_Run  ; Loop3 Process Value, Maximum temperature allowed to run the machine
ANDNOT Tray3_SENSOR_Error  ; Loop3 SENSOR error
ORLD
LD>=(325) Loaded_Recipe_Number_of_Trays &4  ; # of trays in tool
AND>S(322) Tray4_PV Max_Temp_To_Run  ; Loop4 Process Value, Maximum temperature allowed to run the machine
ANDNOT Tray4_SENSOR_Error  ; Loop4 SENSOR error
ORLD
LD>=(325) Loaded_Recipe_Number_of_Trays &5  ; # of trays in tool
AND>S(322) Tray5_PV Max_Temp_To_Run  ; Loop5 Process Value, Maximum temperature allowed to run the machine
ANDNOT Tray5_SENSOR_Error  ; Loop5 SENSOR error
ORLD
LD P_Off
AND=(300) Loaded_Recipe_Number_of_Trays &6  ; # of trays in tool
AND>S(322) NotUsedTray6_PV Max_Temp_To_Run  ; Loop6 Process Value, Maximum temperature allowed to run the machine
ANDNOT NotUsedTray6_SENSOR_Error  ; Loop6 SENSOR error
ORLD
LDNOT Run_latch  ; Machine Run Latch
LD Run_latch  ; Machine Run Latch
@AND Beginning_of_Cycle  ; Beginning of the cycle
ORLD
ANDLD
ANDNOT Sleep_Mode  ; Sleep Mode enabled - drop temp and fault
ANDNOT Upper_Tool_NOT_Locked  ; Upper Tool NOT Locked Bit
TIMHX(551) OverTemp_Delay &200  ; Delay for Over Temperature Fault
AND OverTemp_Delay  ; Delay for Over Temperature Fault
SET Termperature_High  ; Temperature too high enough to run product
; rung 35
LD Sleep_Mode  ; Sleep Mode enabled - drop temp and fault
RSET Teperature_Low  ; Temperature not high enough to run product
RSET Termperature_High  ; Temperature too high enough to run product
; rung 36
LDNOT ipState_AC_Drive_OK  ; AC Drive OK input logical State
OUT AC_Drive_Fault

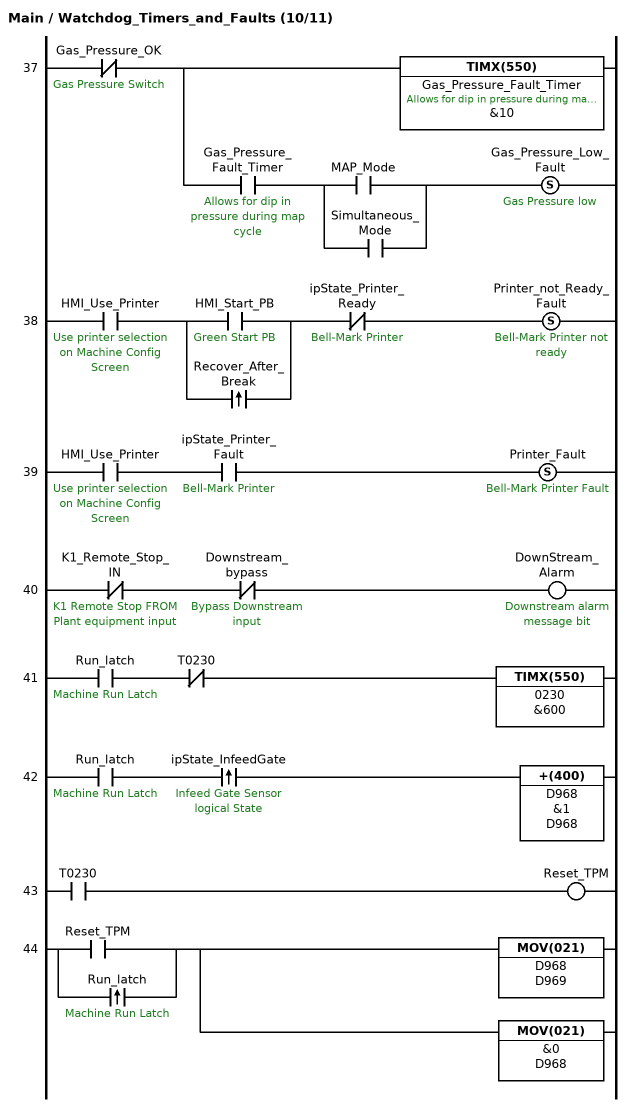
; rung 37
LDNOT Gas_Pressure_OK  ; Gas Pressure Switch
TIMX(550) Gas_Pressure_Fault_Timer &10  ; Allows for dip in pressure during map cycle
AND Gas_Pressure_Fault_Timer  ; Allows for dip in pressure during map cycle
LD MAP_Mode
OR Simultaneous_Mode
ANDLD
SET Gas_Pressure_Low_Fault  ; Gas Pressure low
; rung 38
LD HMI_Use_Printer  ; Use printer selection on Machine Config Screen
LD HMI_Start_PB  ; Green Start PB
@OR Recover_After_Break
ANDLD
ANDNOT ipState_Printer_Ready  ; Bell-Mark Printer
SET Printer_not_Ready_Fault  ; Bell-Mark Printer not ready
; rung 39
LD HMI_Use_Printer  ; Use printer selection on Machine Config Screen
AND ipState_Printer_Fault  ; Bell-Mark Printer
SET Printer_Fault  ; Bell-Mark Printer Fault
; rung 40
LDNOT K1_Remote_Stop_IN  ; K1 Remote Stop FROM Plant equipment input
ANDNOT Downstream_bypass  ; Bypass Downstream input
OUT DownStream_Alarm  ; Downstream alarm message bit
; rung 41
LD Run_latch  ; Machine Run Latch
ANDNOT T0230
TIMX(550) 0230 &600
; rung 42
LD Run_latch  ; Machine Run Latch
@AND ipState_InfeedGate  ; Infeed Gate Sensor logical State
+(400) D968 &1 D968
; rung 43
LD T0230
OUT Reset_TPM
; rung 44
LD Reset_TPM
@OR Run_latch  ; Machine Run Latch
MOV(021) D968 D969
MOV(021) &0 D968

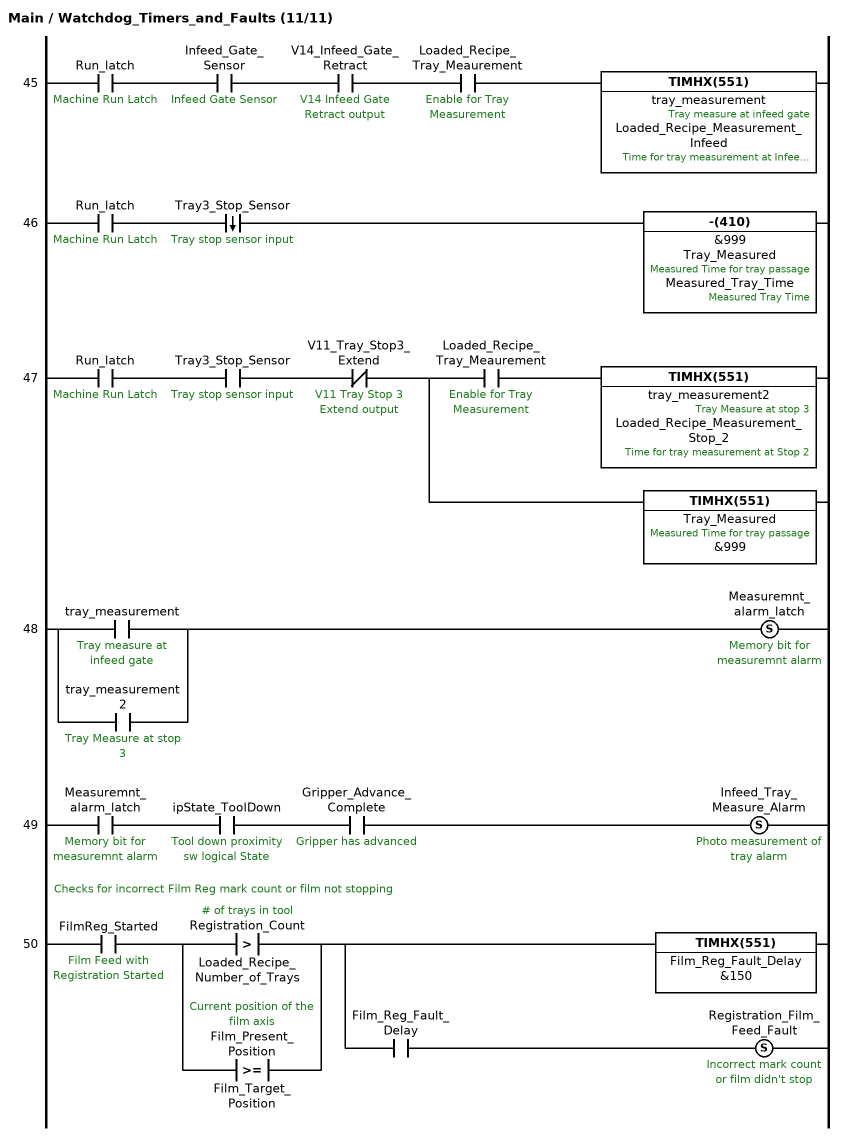
; rung 45
LD Run_latch  ; Machine Run Latch
AND Infeed_Gate_Sensor  ; Infeed Gate Sensor
AND V14_Infeed_Gate_Retract  ; V14 Infeed Gate Retract output
AND Loaded_Recipe_Tray_Meaurement  ; Enable for Tray Measurement
TIMHX(551) tray_measurement Loaded_Recipe_Measurement_Infeed  ; Tray measure at infeed gate, Time for tray measurement at Infeed Gate
; rung 46
LD Run_latch  ; Machine Run Latch
%AND Tray3_Stop_Sensor  ; Tray stop sensor input
-(410) &999 Tray_Measured Measured_Tray_Time  ; Measured Time for tray passage, Measured Tray Time
; rung 47
LD Run_latch  ; Machine Run Latch
AND Tray3_Stop_Sensor  ; Tray stop sensor input
ANDNOT V11_Tray_Stop3_Extend  ; V11 Tray Stop 3 Extend output
OUT TR0
AND Loaded_Recipe_Tray_Meaurement  ; Enable for Tray Measurement
TIMHX(551) tray_measurement2 Loaded_Recipe_Measurement_Stop_2  ; Tray Measure at stop 3, Time for tray measurement at Stop 2
LD TR0
TIMHX(551) Tray_Measured &999  ; Measured Time for tray passage
; rung 48
LD tray_measurement  ; Tray measure at infeed gate
OR tray_measurement2  ; Tray Measure at stop 3
SET Measuremnt_alarm_latch  ; Memory bit for measuremnt alarm
; rung 49
LD Measuremnt_alarm_latch  ; Memory bit for measuremnt alarm
AND ipState_ToolDown  ; Tool down proximity sw logical State
AND Gripper_Advance_Complete  ; Gripper has advanced
SET Infeed_Tray_Measure_Alarm  ; Photo measurement of tray alarm
; rung 50: Checks for incorrect Film Reg mark count or film not stopping
LD FilmReg_Started  ; Film Feed with Registration Started
LD>(320) Registration_Count Loaded_Recipe_Number_of_Trays  ; # of trays in tool
OR>=(325) Film_Present_Position Film_Target_Position  ; Current position of the film axis
ANDLD
TIMHX(551) Film_Reg_Fault_Delay &150
AND Film_Reg_Fault_Delay
SET Registration_Film_Feed_Fault  ; Incorrect mark count or film didn't stop

### Section Gripper_Servo

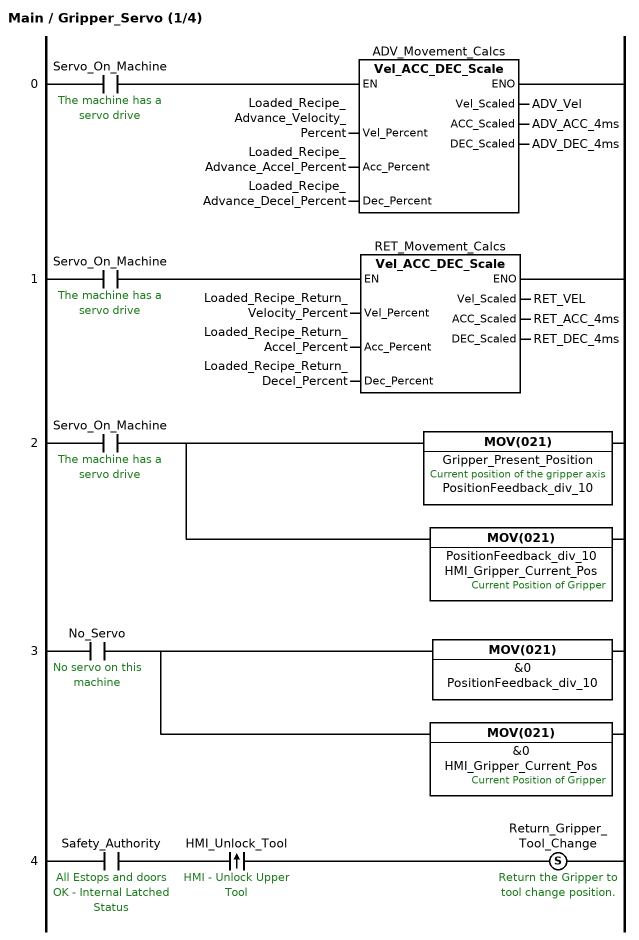
; rung 0
LD Servo_On_Machine  ; The machine has a servo drive
CALL ADV_Movement_Calcs : Vel_ACC_DEC_Scale (Vel_Percent := Loaded_Recipe_Advance_Velocity_Percent, Acc_Percent := Loaded_Recipe_Advance_Accel_Percent, Dec_Percent := Loaded_Recipe_Advance_Decel_Percent, Vel_Scaled => ADV_Vel, ACC_Scaled => ADV_ACC_4ms, DEC_Scaled => ADV_DEC_4ms)
; rung 1
LD Servo_On_Machine  ; The machine has a servo drive
CALL RET_Movement_Calcs : Vel_ACC_DEC_Scale (Vel_Percent := Loaded_Recipe_Return_Velocity_Percent, Acc_Percent := Loaded_Recipe_Return_Accel_Percent, Dec_Percent := Loaded_Recipe_Return_Decel_Percent, Vel_Scaled => RET_VEL, ACC_Scaled => RET_ACC_4ms, DEC_Scaled => RET_DEC_4ms)
; rung 2
LD Servo_On_Machine  ; The machine has a servo drive
MOV(021) Gripper_Present_Position PositionFeedback_div_10  ; Current position of the gripper axis
MOV(021) PositionFeedback_div_10 HMI_Gripper_Current_Pos  ; Current Position of Gripper
; rung 3
LD No_Servo  ; No servo on this machine
MOV(021) &0 PositionFeedback_div_10
MOV(021) &0 HMI_Gripper_Current_Pos  ; Current Position of Gripper
; rung 4
LD Safety_Authority  ; All Estops and doors OK - Internal Latched Status
@AND HMI_Unlock_Tool  ; HMI - Unlock Upper Tool
SET Return_Gripper_Tool_Change  ; Return the Gripper to tool change position.

